LIN {X 0,Y 362.029,Z 234.39,A -85,B 0,C 180,E1 -12949.938,E2 -12949.938} C_VEL
LIN {X 0,Y 362.149,Z 234.377,A -85,B 0,C 180,E1 -12952.192,E2 -12952.192} C_VEL
LIN {X 0,Y 362.116,Z 234.379,A -85,B 0,C 180,E1 -12954.431,E2 -12954.431} C_VEL
LIN {X 0,Y 362.28,Z 234.357,A -85,B 0,C 180,E1 -12957.776,E2 -12957.776} C_VEL
LIN {X 0,Y 362.423,Z 234.341,A -85,B 0,C 180,E1 -12960,E2 -12960} C_VEL
LIN {X 0,Y 362.28,Z 234.36,A -85,B 0,C 180,E1 -12962.223,E2 -12962.223} C_VEL
LIN {X 0,Y 362.17,Z 234.37,A -85,B 0,C 180,E1 -12966.686,E2 -12966.686} C_VEL
LIN {X 0,Y 362.071,Z 234.381,A -85,B 0,C 180,E1 -12968.933,E2 -12968.933} C_VEL
LIN {X 0,Y 361.958,Z 234.4,A -85,B 0,C 180,E1 -12972.332,E2 -12972.332} C_VEL
LIN {X 0,Y 361.959,Z 234.397,A -85,B 0,C 180,E1 -12974.62,E2 -12974.62} C_VEL
LIN {X 0,Y 361.957,Z 234.4,A -85,B 0,C 180,E1 -12978.099,E2 -12978.099} C_VEL
LIN {X 0,Y 361.89,Z 234.404,A -85,B 0,C 180,E1 -12981.653,E2 -12981.653} C_VEL
LIN {X 0,Y 361.926,Z 234.399,A -85,B 0,C 180,E1 -12985.29,E2 -12985.29} C_VEL
LIN {X 0,Y 361.916,Z 234.401,A -85,B 0,C 180,E1 -12987.778,E2 -12987.778} C_VEL
LIN {X 0,Y 361.844,Z 234.409,A -85,B 0,C 180,E1 -12991.285,E2 -12991.285} C_VEL
LIN {X 0,Y 361.852,Z 234.413,A -85,B 0,C 180,E1 -12994.281,E2 -12994.281} C_VEL
LIN {X 0,Y 361.862,Z 234.407,A -85,B 0,C 180,E1 -12997.223,E2 -12997.223} C_VEL
LIN {X 0,Y 361.834,Z 234.413,A -85,B 0,C 180,E1 -13000.756,E2 -13000.756} C_VEL
LIN {X 0,Y 361.816,Z 234.418,A -85,B 0,C 180,E1 -13004.369,E2 -13004.369} C_VEL
LIN {X 0,Y 361.835,Z 234.41,A -85,B 0,C 180,E1 -13007.568,E2 -13007.568} C_VEL
LIN {X 0,Y 361.869,Z 234.407,A -85,B 0,C 180,E1 -13010.974,E2 -13010.974} C_VEL
LIN {X 0,Y 361.874,Z 234.409,A -85,B 0,C 180,E1 -13014.656,E2 -13014.656} C_VEL
LIN {X 0,Y 361.838,Z 234.415,A -85,B 0,C 180,E1 -13018.371,E2 -13018.371} C_VEL
LIN {X 0,Y 361.919,Z 234.533,A -85,B 0,C 180,E1 -13020.495,E2 -13020.495} C_VEL
LIN {X 0,Y 364.089,Z 244.857,A -85,B 0,C 180,E1 -13023.197,E2 -13023.197} C_VEL
LIN {X 0,Y 365.508,Z 253.131,A -85,B 0,C 180,E1 -13025.279,E2 -13025.279} C_VEL
LIN {X 0,Y 364.772,Z 261.991,A -85,B 0,C 180,E1 -13027.336,E2 -13027.336} C_VEL
LIN {X 0,Y 364.414,Z 265.703,A -85,B 0,C 180,E1 -13028.19,E2 -13028.19} C_VEL
LIN {X 0,Y 369.621,Z 298.526,A -85,B 0,C 180,E1 -13029.181,E2 -13029.181} C_VEL
LIN {X 0,Y 368.296,Z 374.24,A -85,B 0,C 180,E1 -13030.709,E2 -13030.709} C_VEL
LIN {X 0,Y 367.689,Z 387.314,A -85,B 0,C 180,E1 -13031.183,E2 -13031.183} C_VEL
LIN {X 0,Y 366.8,Z 399.96,A -85,B 0,C 180,E1 -13031.859,E2 -13031.859} C_VEL
LIN {X 0,Y 365.939,Z 411.236,A -85,B 0,C 180,E1 -13032.682,E2 -13032.682} C_VEL
LIN {X 0,Y 364.86,Z 422.904,A -85,B 0,C 180,E1 -13033.782,E2 -13033.782} C_VEL
LIN {X 0,Y 363.982,Z 432.341,A -85,B 0,C 180,E1 -13034.892,E2 -13034.892} C_VEL
LIN {X 0,Y 363.055,Z 441.998,A -85,B 0,C 180,E1 -13036.283,E2 -13036.283} C_VEL
LIN {X 0,Y 362.203,Z 449.91,A -85,B 0,C 180,E1 -13037.676,E2 -13037.676} C_VEL
LIN {X 0,Y 361.425,Z 457.628,A -85,B 0,C 180,E1 -13039.355,E2 -13039.355} C_VEL
LIN {X 0,Y 360.913,Z 463.827,A -85,B 0,C 180,E1 -13041.038,E2 -13041.038} C_VEL
LIN {X 0,Y 360.588,Z 468.742,A -85,B 0,C 180,E1 -13042.722,E2 -13042.722} C_VEL
LIN {X 0,Y 360.383,Z 472.518,A -85,B 0,C 180,E1 -13044.405,E2 -13044.405} C_VEL
LIN {X 0,Y 360.364,Z 474.464,A -85,B 0,C 180,E1 -13045.526,E2 -13045.526} C_VEL
LIN {X 0,Y 360.3,Z 475.982,A -85,B 0,C 180,E1 -13046.645,E2 -13046.645} C_VEL
LIN {X 0,Y 360.317,Z 477.708,A -85,B 0,C 180,E1 -13048.883,E2 -13048.883} C_VEL
LIN {X 0,Y 360.359,Z 477.984,A -85,B 0,C 180,E1 -13050,E2 -13050} C_VEL
LIN {X 0,Y 360.302,Z 477.86,A -85,B 0,C 180,E1 -13051.118,E2 -13051.118} C_VEL
LIN {X 0,Y 360.297,Z 476.346,A -85,B 0,C 180,E1 -13053.355,E2 -13053.355} C_VEL
LIN {X 0,Y 360.347,Z 474.995,A -85,B 0,C 180,E1 -13054.475,E2 -13054.475} C_VEL
LIN {X 0,Y 360.378,Z 472.521,A -85,B 0,C 180,E1 -13055.961,E2 -13055.961} C_VEL
LIN {X 0,Y 360.672,Z 468.262,A -85,B 0,C 180,E1 -13057.84,E2 -13057.84} C_VEL
LIN {X 0,Y 361.092,Z 463.255,A -85,B 0,C 180,E1 -13059.523,E2 -13059.523} C_VEL
LIN {X 0,Y 361.706,Z 456.971,A -85,B 0,C 180,E1 -13061.204,E2 -13061.204} C_VEL
LIN {X 0,Y 362.689,Z 449.128,A -85,B 0,C 180,E1 -13062.876,E2 -13062.876} C_VEL
LIN {X 0,Y 363.572,Z 441.13,A -85,B 0,C 180,E1 -13064.268,E2 -13064.268} C_VEL
LIN {X 0,Y 364.586,Z 431.385,A -85,B 0,C 180,E1 -13065.657,E2 -13065.657} C_VEL
LIN {X 0,Y 365.793,Z 420.582,A -85,B 0,C 180,E1 -13066.894,E2 -13066.894} C_VEL
LIN {X 0,Y 366.82,Z 410.08,A -85,B 0,C 180,E1 -13067.851,E2 -13067.851} C_VEL
LIN {X 0,Y 367.955,Z 397.467,A -85,B 0,C 180,E1 -13068.731,E2 -13068.731} C_VEL
LIN {X 0,Y 368.842,Z 384.167,A -85,B 0,C 180,E1 -13069.406,E2 -13069.406} C_VEL
LIN {X 0,Y 369.489,Z 370.423,A -85,B 0,C 180,E1 -13069.841,E2 -13069.841} C_VEL
LIN {X 0,Y 370.705,Z 298.181,A -85,B 0,C 180,E1 -13071.303,E2 -13071.303} C_VEL
LIN {X 0,Y 366.607,Z 273.496,A -85,B 0,C 180,E1 -13072.105,E2 -13072.105} C_VEL
LIN {X 0,Y 364.918,Z 264.825,A -85,B 0,C 180,E1 -13072.438,E2 -13072.438} C_VEL
LIN {X 0,Y 365.842,Z 254.94,A -85,B 0,C 180,E1 -13074.698,E2 -13074.698} C_VEL
LIN {X 0,Y 365.142,Z 249.633,A -85,B 0,C 180,E1 -13076.012,E2 -13076.012} C_VEL
LIN {X 0,Y 363.099,Z 239.586,A -85,B 0,C 180,E1 -13078.623,E2 -13078.623} C_VEL
LIN {X 0,Y 361.883,Z 234.409,A -85,B 0,C 180,E1 -13080.023,E2 -13080.023} C_VEL
LIN {X 0,Y 361.86,Z 234.415,A -85,B 0,C 180,E1 -13083.369,E2 -13083.369} C_VEL
LIN {X 0,Y 361.867,Z 234.412,A -85,B 0,C 180,E1 -13087.018,E2 -13087.018} C_VEL
LIN {X 0,Y 361.855,Z 234.408,A -85,B 0,C 180,E1 -13089.861,E2 -13089.861} C_VEL
LIN {X 0,Y 361.837,Z 234.411,A -85,B 0,C 180,E1 -13092.829,E2 -13092.829} C_VEL
LIN {X 0,Y 361.819,Z 234.416,A -85,B 0,C 180,E1 -13095.946,E2 -13095.946} C_VEL
LIN {X 0,Y 361.836,Z 234.415,A -85,B 0,C 180,E1 -13099.244,E2 -13099.244} C_VEL
LIN {X 0,Y 361.863,Z 234.409,A -85,B 0,C 180,E1 -13102.777,E2 -13102.777} C_VEL
LIN {X 0,Y 361.854,Z 234.409,A -85,B 0,C 180,E1 -13105.72,E2 -13105.72} C_VEL
LIN {X 0,Y 361.872,Z 234.407,A -85,B 0,C 180,E1 -13109.672,E2 -13109.672} C_VEL
LIN {X 0,Y 361.954,Z 234.396,A -85,B 0,C 180,E1 -13113.475,E2 -13113.475} C_VEL
LIN {X 0,Y 361.89,Z 234.401,A -85,B 0,C 180,E1 -13117.145,E2 -13117.145} C_VEL
LIN {X 0,Y 361.92,Z 234.399,A -85,B 0,C 180,E1 -13120.724,E2 -13120.724} C_VEL
LIN {X 0,Y 361.945,Z 234.397,A -85,B 0,C 180,E1 -13124.226,E2 -13124.226} C_VEL
LIN {X 0,Y 361.998,Z 234.383,A -85,B 0,C 180,E1 -13126.528,E2 -13126.528} C_VEL
LIN {X 0,Y 362.031,Z 234.381,A -85,B 0,C 180,E1 -13129.938,E2 -13129.938} C_VEL
LIN {X 0,Y 362.16,Z 234.371,A -85,B 0,C 180,E1 -13133.314,E2 -13133.314} C_VEL
LIN {X 0,Y 362.282,Z 234.355,A -85,B 0,C 180,E1 -13137.777,E2 -13137.777} C_VEL
LIN {X 0,Y 362.426,Z 234.33,A -85,B 0,C 180,E1 -13140,E2 -13140} C_VEL
LIN {X 0,Y 362.281,Z 234.357,A -85,B 0,C 180,E1 -13142.224,E2 -13142.224} C_VEL
LIN {X 0,Y 362.17,Z 234.372,A -85,B 0,C 180,E1 -13146.686,E2 -13146.686} C_VEL
LIN {X 0,Y 362.074,Z 234.382,A -85,B 0,C 180,E1 -13148.933,E2 -13148.933} C_VEL
LIN {X 0,Y 361.959,Z 234.392,A -85,B 0,C 180,E1 -13152.332,E2 -13152.332} C_VEL
LIN {X 0,Y 361.962,Z 234.396,A -85,B 0,C 180,E1 -13154.621,E2 -13154.621} C_VEL
LIN {X 0,Y 361.96,Z 234.396,A -85,B 0,C 180,E1 -13158.099,E2 -13158.099} C_VEL
LIN {X 0,Y 361.861,Z 234.408,A -85,B 0,C 180,E1 -13161.655,E2 -13161.655} C_VEL
LIN {X 0,Y 361.901,Z 234.405,A -85,B 0,C 180,E1 -13165.292,E2 -13165.292} C_VEL
LIN {X 0,Y 361.874,Z 234.4,A -85,B 0,C 180,E1 -13169.079,E2 -13169.079} C_VEL
LIN {X 0,Y 361.848,Z 234.411,A -85,B 0,C 180,E1 -13172.945,E2 -13172.945} C_VEL
LIN {X 0,Y 361.867,Z 234.412,A -85,B 0,C 180,E1 -13175.637,E2 -13175.637} C_VEL
LIN {X 0,Y 361.876,Z 234.589,A -85,B 0,C 180,E1 -13179.214,E2 -13179.214} C_VEL
LIN {X 0,Y 364.197,Z 245.232,A -85,B 0,C 180,E1 -13182.112,E2 -13182.112} C_VEL
LIN {X 0,Y 364.641,Z 247.353,A -85,B 0,C 180,E1 -13182.626,E2 -13182.626} C_VEL
LIN {X 0,Y 367.364,Z 255.054,A -85,B 0,C 180,E1 -13182.986,E2 -13182.986} C_VEL
LIN {X 0,Y 371.258,Z 274.03,A -85,B 0,C 180,E1 -13183.657,E2 -13183.657} C_VEL
LIN {X 0,Y 369.515,Z 355.097,A -85,B 0,C 180,E1 -13185.298,E2 -13185.298} C_VEL
LIN {X 0,Y 368.933,Z 368.742,A -85,B 0,C 180,E1 -13185.807,E2 -13185.807} C_VEL
LIN {X 0,Y 368.181,Z 381.251,A -85,B 0,C 180,E1 -13186.499,E2 -13186.499} C_VEL
LIN {X 0,Y 367.234,Z 393.083,A -85,B 0,C 180,E1 -13187.391,E2 -13187.391} C_VEL
LIN {X 0,Y 366.107,Z 405.138,A -85,B 0,C 180,E1 -13188.568,E2 -13188.568} C_VEL
LIN {X 0,Y 364.993,Z 415.361,A -85,B 0,C 180,E1 -13189.832,E2 -13189.832} C_VEL
LIN {X 0,Y 363.968,Z 423.909,A -85,B 0,C 180,E1 -13191.13,E2 -13191.13} C_VEL
LIN {X 0,Y 362.95,Z 432.857,A -85,B 0,C 180,E1 -13192.811,E2 -13192.811} C_VEL
LIN {X 0,Y 362.12,Z 439.647,A -85,B 0,C 180,E1 -13194.392,E2 -13194.392} C_VEL
LIN {X 0,Y 361.357,Z 446.052,A -85,B 0,C 180,E1 -13196.277,E2 -13196.277} C_VEL
LIN {X 0,Y 360.866,Z 451.154,A -85,B 0,C 180,E1 -13198.276,E2 -13198.276} C_VEL
LIN {X 0,Y 360.624,Z 453.662,A -85,B 0,C 180,E1 -13199.556,E2 -13199.556} C_VEL
LIN {X 0,Y 360.339,Z 456.193,A -85,B 0,C 180,E1 -13201.364,E2 -13201.364} C_VEL
LIN {X 0,Y 360.124,Z 457.717,A -85,B 0,C 180,E1 -13203.33,E2 -13203.33} C_VEL
LIN {X 0,Y 360.085,Z 458.053,A -85,B 0,C 180,E1 -13204.571,E2 -13204.571} C_VEL
LIN {X 0,Y 360.06,Z 457.594,A -85,B 0,C 180,E1 -13206.549,E2 -13206.549} C_VEL
LIN {X 0,Y 360.208,Z 456.184,A -85,B 0,C 180,E1 -13208.241,E2 -13208.241} C_VEL
LIN {X 0,Y 360.519,Z 453.638,A -85,B 0,C 180,E1 -13210.053,E2 -13210.053} C_VEL
LIN {X 0,Y 360.83,Z 449.998,A -85,B 0,C 180,E1 -13211.842,E2 -13211.842} C_VEL
LIN {X 0,Y 361.209,Z 445.164,A -85,B 0,C 180,E1 -13213.613,E2 -13213.613} C_VEL
LIN {X 0,Y 361.808,Z 438.966,A -85,B 0,C 180,E1 -13215.373,E2 -13215.373} C_VEL
LIN {X 0,Y 362.631,Z 431.207,A -85,B 0,C 180,E1 -13217.122,E2 -13217.122} C_VEL
LIN {X 0,Y 363.465,Z 423.268,A -85,B 0,C 180,E1 -13218.568,E2 -13218.568} C_VEL
LIN {X 0,Y 364.469,Z 413.538,A -85,B 0,C 180,E1 -13220.006,E2 -13220.006} C_VEL
LIN {X 0,Y 365.519,Z 402.66,A -85,B 0,C 180,E1 -13221.291,E2 -13221.291} C_VEL
LIN {X 0,Y 366.484,Z 392.105,A -85,B 0,C 180,E1 -13222.285,E2 -13222.285} C_VEL
LIN {X 0,Y 367.251,Z 380.768,A -85,B 0,C 180,E1 -13223.131,E2 -13223.131} C_VEL
LIN {X 0,Y 367.916,Z 368.075,A -85,B 0,C 180,E1 -13223.828,E2 -13223.828} C_VEL
LIN {X 0,Y 368.443,Z 354.712,A -85,B 0,C 180,E1 -13224.321,E2 -13224.321} C_VEL
LIN {X 0,Y 369.856,Z 272.512,A -85,B 0,C 180,E1 -13225.982,E2 -13225.982} C_VEL
LIN {X 0,Y 365.244,Z 249.773,A -85,B 0,C 180,E1 -13226.725,E2 -13226.725} C_VEL
LIN {X 0,Y 364.343,Z 246.957,A -85,B 0,C 180,E1 -13226.855,E2 -13226.855} C_VEL
LIN {X 0,Y 363.165,Z 239.521,A -85,B 0,C 180,E1 -13228.891,E2 -13228.891} C_VEL
LIN {X 0,Y 362.19,Z 234.367,A -85,B 0,C 180,E1 -13230.347,E2 -13230.347} C_VEL
LIN {X 0,Y 362.268,Z 234.36,A -85,B 0,C 180,E1 -13232.223,E2 -13232.223} C_VEL
LIN {X 0,Y 362.125,Z 234.374,A -85,B 0,C 180,E1 -13236.687,E2 -13236.687} C_VEL
LIN {X 0,Y 362.048,Z 234.383,A -85,B 0,C 180,E1 -13238.934,E2 -13238.934} C_VEL
LIN {X 0,Y 361.325,Z 234.479,A -85,B 0,C 180,E1 -13239.862,E2 -13239.862} C_VEL
LIN {X 0,Y 358.466,Z 234.835,A -85,B 0,C 180,E1 -13241.37,E2 -13241.37} C_VEL
LIN {X 0,Y 356.073,Z 235.136,A -85,B 0,C 180,E1 -13242.59,E2 -13242.59} C_VEL
LIN {X 0,Y 355.039,Z 235.263,A -85,B 0,C 180,E1 -13243.534,E2 -13243.534} C_VEL
LIN {X 0,Y 354.95,Z 235.272,A -85,B 0,C 180,E1 -13243.853,E2 -13243.853} C_VEL
LIN {X 0,Y 354.925,Z 235.274,A -85,B 0,C 180,E1 -13248.108,E2 -13248.108} C_VEL
LIN {X 0,Y 354.828,Z 235.286,A -85,B 0,C 180,E1 -13252.106,E2 -13252.106} C_VEL
LIN {X 0,Y 354.852,Z 235.286,A -85,B 0,C 180,E1 -13255.831,E2 -13255.831} C_VEL
LIN {X 0,Y 354.8,Z 235.29,A -85,B 0,C 180,E1 -13259.683,E2 -13259.683} C_VEL
LIN {X 0,Y 354.788,Z 235.29,A -85,B 0,C 180,E1 -13262.333,E2 -13262.333} C_VEL
LIN {X 0,Y 354.822,Z 235.288,A -85,B 0,C 180,E1 -13265.699,E2 -13265.699} C_VEL
LIN {X 0,Y 354.824,Z 235.285,A -85,B 0,C 180,E1 -13269.423,E2 -13269.423} C_VEL
LIN {X 0,Y 354.786,Z 235.288,A -85,B 0,C 180,E1 -13272.866,E2 -13272.866} C_VEL
LIN {X 0,Y 354.766,Z 235.295,A -85,B 0,C 180,E1 -13276.103,E2 -13276.103} C_VEL
LIN {X 0,Y 354.786,Z 235.288,A -85,B 0,C 180,E1 -13279.178,E2 -13279.178} C_VEL
LIN {X 0,Y 354.806,Z 235.288,A -85,B 0,C 180,E1 -13282.402,E2 -13282.402} C_VEL
LIN {X 0,Y 354.81,Z 235.285,A -85,B 0,C 180,E1 -13284.94,E2 -13284.94} C_VEL
LIN {X 0,Y 354.792,Z 235.29,A -85,B 0,C 180,E1 -13288.405,E2 -13288.405} C_VEL
LIN {X 0,Y 354.845,Z 235.283,A -85,B 0,C 180,E1 -13291.618,E2 -13291.618} C_VEL
LIN {X 0,Y 354.897,Z 235.279,A -85,B 0,C 180,E1 -13294.172,E2 -13294.172} C_VEL
LIN {X 0,Y 354.833,Z 235.287,A -85,B 0,C 180,E1 -13297.894,E2 -13297.894} C_VEL
LIN {X 0,Y 354.92,Z 235.276,A -85,B 0,C 180,E1 -13301.891,E2 -13301.891} C_VEL
LIN {X 0,Y 354.94,Z 235.274,A -85,B 0,C 180,E1 -13305.981,E2 -13305.981} C_VEL
LIN {X 0,Y 354.976,Z 235.267,A -85,B 0,C 180,E1 -13309.736,E2 -13309.736} C_VEL
LIN {X 0,Y 355.112,Z 235.253,A -85,B 0,C 180,E1 -13312.037,E2 -13312.037} C_VEL
LIN {X 0,Y 355.09,Z 235.255,A -85,B 0,C 180,E1 -13314.321,E2 -13314.321} C_VEL
LIN {X 0,Y 355.243,Z 235.233,A -85,B 0,C 180,E1 -13317.732,E2 -13317.732} C_VEL
LIN {X 0,Y 355.393,Z 235.217,A -85,B 0,C 180,E1 -13320,E2 -13320} C_VEL
LIN {X 0,Y 355.243,Z 235.237,A -85,B 0,C 180,E1 -13322.268,E2 -13322.268} C_VEL
LIN {X 0,Y 355.136,Z 235.245,A -85,B 0,C 180,E1 -13326.819,E2 -13326.819} C_VEL
LIN {X 0,Y 355.013,Z 235.26,A -85,B 0,C 180,E1 -13329.112,E2 -13329.112} C_VEL
LIN {X 0,Y 354.919,Z 235.274,A -85,B 0,C 180,E1 -13332.581,E2 -13332.581} C_VEL
LIN {X 0,Y 354.887,Z 235.28,A -85,B 0,C 180,E1 -13336.096,E2 -13336.096} C_VEL
LIN {X 0,Y 354.904,Z 235.278,A -85,B 0,C 180,E1 -13338.472,E2 -13338.472} C_VEL
LIN {X 0,Y 354.832,Z 235.287,A -85,B 0,C 180,E1 -13342.106,E2 -13342.106} C_VEL
LIN {X 0,Y 354.897,Z 235.276,A -85,B 0,C 180,E1 -13345.828,E2 -13345.828} C_VEL
LIN {X 0,Y 354.852,Z 235.28,A -85,B 0,C 180,E1 -13349.679,E2 -13349.679} C_VEL
LIN {X 0,Y 354.804,Z 235.286,A -85,B 0,C 180,E1 -13353.702,E2 -13353.702} C_VEL
LIN {X 0,Y 354.797,Z 235.292,A -85,B 0,C 180,E1 -13356.46,E2 -13356.46} C_VEL
LIN {X 0,Y 354.822,Z 235.283,A -85,B 0,C 180,E1 -13359.424,E2 -13359.424} C_VEL
LIN {X 0,Y 354.786,Z 235.29,A -85,B 0,C 180,E1 -13362.868,E2 -13362.868} C_VEL
LIN {X 0,Y 354.766,Z 235.294,A -85,B 0,C 180,E1 -13366.104,E2 -13366.104} C_VEL
LIN {X 0,Y 354.787,Z 235.288,A -85,B 0,C 180,E1 -13369.179,E2 -13369.179} C_VEL
LIN {X 0,Y 354.81,Z 235.291,A -85,B 0,C 180,E1 -13372.402,E2 -13372.402} C_VEL
LIN {X 0,Y 354.811,Z 235.286,A -85,B 0,C 180,E1 -13374.941,E2 -13374.941} C_VEL
LIN {X 0,Y 354.793,Z 235.293,A -85,B 0,C 180,E1 -13378.405,E2 -13378.405} C_VEL
LIN {X 0,Y 354.871,Z 235.377,A -85,B 0,C 180,E1 -13380.16,E2 -13380.16} C_VEL
LIN {X 0,Y 357.175,Z 246.354,A -85,B 0,C 180,E1 -13383.092,E2 -13383.092} C_VEL
LIN {X 0,Y 358.515,Z 254.059,A -85,B 0,C 180,E1 -13385.073,E2 -13385.073} C_VEL
LIN {X 0,Y 357.995,Z 261.662,A -85,B 0,C 180,E1 -13386.882,E2 -13386.882} C_VEL
LIN {X 0,Y 357.535,Z 265.52,A -85,B 0,C 180,E1 -13387.783,E2 -13387.783} C_VEL
LIN {X 0,Y 362.845,Z 298.374,A -85,B 0,C 180,E1 -13388.804,E2 -13388.804} C_VEL
LIN {X 0,Y 361.735,Z 368.666,A -85,B 0,C 180,E1 -13390.234,E2 -13390.234} C_VEL
LIN {X 0,Y 361.18,Z 382.385,A -85,B 0,C 180,E1 -13390.646,E2 -13390.646} C_VEL
LIN {X 0,Y 360.411,Z 394.736,A -85,B 0,C 180,E1 -13391.232,E2 -13391.232} C_VEL
LIN {X 0,Y 359.636,Z 405.389,A -85,B 0,C 180,E1 -13391.927,E2 -13391.927} C_VEL
LIN {X 0,Y 358.569,Z 416.918,A -85,B 0,C 180,E1 -13392.903,E2 -13392.903} C_VEL
LIN {X 0,Y 357.4,Z 428.473,A -85,B 0,C 180,E1 -13394.153,E2 -13394.153} C_VEL
LIN {X 0,Y 356.531,Z 438.002,A -85,B 0,C 180,E1 -13395.444,E2 -13395.444} C_VEL
LIN {X 0,Y 355.606,Z 446.571,A -85,B 0,C 180,E1 -13396.863,E2 -13396.863} C_VEL
LIN {X 0,Y 354.604,Z 454.901,A -85,B 0,C 180,E1 -13398.569,E2 -13398.569} C_VEL
LIN {X 0,Y 354.018,Z 461.619,A -85,B 0,C 180,E1 -13400.286,E2 -13400.286} C_VEL
LIN {X 0,Y 353.609,Z 466.972,A -85,B 0,C 180,E1 -13402.003,E2 -13402.003} C_VEL
LIN {X 0,Y 353.314,Z 471.786,A -85,B 0,C 180,E1 -13404.035,E2 -13404.035} C_VEL
LIN {X 0,Y 353.277,Z 474.224,A -85,B 0,C 180,E1 -13405.436,E2 -13405.436} C_VEL
LIN {X 0,Y 353.222,Z 475.755,A -85,B 0,C 180,E1 -13406.578,E2 -13406.578} C_VEL
LIN {X 0,Y 353.217,Z 477.5,A -85,B 0,C 180,E1 -13408.86,E2 -13408.86} C_VEL
LIN {X 0,Y 353.262,Z 477.783,A -85,B 0,C 180,E1 -13410,E2 -13410} C_VEL
LIN {X 0,Y 353.202,Z 477.67,A -85,B 0,C 180,E1 -13411.14,E2 -13411.14} C_VEL
LIN {X 0,Y 353.171,Z 477.121,A -85,B 0,C 180,E1 -13412.281,E2 -13412.281} C_VEL
LIN {X 0,Y 353.218,Z 476.174,A -85,B 0,C 180,E1 -13413.422,E2 -13413.422} C_VEL
LIN {X 0,Y 353.26,Z 474.829,A -85,B 0,C 180,E1 -13414.564,E2 -13414.564} C_VEL
LIN {X 0,Y 353.275,Z 472.703,A -85,B 0,C 180,E1 -13415.905,E2 -13415.905} C_VEL
LIN {X 0,Y 353.617,Z 468.125,A -85,B 0,C 180,E1 -13417.997,E2 -13417.997} C_VEL
LIN {X 0,Y 354.057,Z 463.133,A -85,B 0,C 180,E1 -13419.714,E2 -13419.714} C_VEL
LIN {X 0,Y 354.704,Z 456.869,A -85,B 0,C 180,E1 -13421.428,E2 -13421.428} C_VEL
LIN {X 0,Y 355.743,Z 449.067,A -85,B 0,C 180,E1 -13423.132,E2 -13423.132} C_VEL
LIN {X 0,Y 356.653,Z 441.105,A -85,B 0,C 180,E1 -13424.551,E2 -13424.551} C_VEL
LIN {X 0,Y 357.881,Z 430.336,A -85,B 0,C 180,E1 -13426.104,E2 -13426.104} C_VEL
LIN {X 0,Y 359.116,Z 419.292,A -85,B 0,C 180,E1 -13427.364,E2 -13427.364} C_VEL
LIN {X 0,Y 360.277,Z 408.49,A -85,B 0,C 180,E1 -13428.334,E2 -13428.334} C_VEL
LIN {X 0,Y 361.361,Z 396.619,A -85,B 0,C 180,E1 -13429.159,E2 -13429.159} C_VEL
LIN {X 0,Y 362.214,Z 383.848,A -85,B 0,C 180,E1 -13429.813,E2 -13429.813} C_VEL
LIN {X 0,Y 362.886,Z 370.019,A -85,B 0,C 180,E1 -13430.254,E2 -13430.254} C_VEL
LIN {X 0,Y 364.227,Z 299.716,A -85,B 0,C 180,E1 -13431.697,E2 -13431.697} C_VEL
LIN {X 0,Y 360.413,Z 276.099,A -85,B 0,C 180,E1 -13432.48,E2 -13432.48} C_VEL
LIN {X 0,Y 358.119,Z 264.715,A -85,B 0,C 180,E1 -13432.905,E2 -13432.905} C_VEL
LIN {X 0,Y 358.954,Z 256.182,A -85,B 0,C 180,E1 -13434.895,E2 -13434.895} C_VEL
LIN {X 0,Y 357.778,Z 248.514,A -85,B 0,C 180,E1 -13436.859,E2 -13436.859} C_VEL
LIN {X 0,Y 355.535,Z 238.291,A -85,B 0,C 180,E1 -13439.616,E2 -13439.616} C_VEL
LIN {X 0,Y 354.84,Z 235.286,A -85,B 0,C 180,E1 -13440.499,E2 -13440.499} C_VEL
LIN {X 0,Y 354.807,Z 235.293,A -85,B 0,C 180,E1 -13443.702,E2 -13443.702} C_VEL
LIN {X 0,Y 354.798,Z 235.289,A -85,B 0,C 180,E1 -13446.459,E2 -13446.459} C_VEL
LIN {X 0,Y 354.825,Z 235.286,A -85,B 0,C 180,E1 -13449.423,E2 -13449.423} C_VEL
LIN {X 0,Y 354.789,Z 235.289,A -85,B 0,C 180,E1 -13452.867,E2 -13452.867} C_VEL
LIN {X 0,Y 354.768,Z 235.294,A -85,B 0,C 180,E1 -13456.104,E2 -13456.104} C_VEL
LIN {X 0,Y 354.788,Z 235.292,A -85,B 0,C 180,E1 -13459.179,E2 -13459.179} C_VEL
LIN {X 0,Y 354.807,Z 235.286,A -85,B 0,C 180,E1 -13462.402,E2 -13462.402} C_VEL
LIN {X 0,Y 354.812,Z 235.283,A -85,B 0,C 180,E1 -13464.941,E2 -13464.941} C_VEL
LIN {X 0,Y 354.793,Z 235.284,A -85,B 0,C 180,E1 -13468.405,E2 -13468.405} C_VEL
LIN {X 0,Y 354.846,Z 235.279,A -85,B 0,C 180,E1 -13471.619,E2 -13471.619} C_VEL
LIN {X 0,Y 354.899,Z 235.274,A -85,B 0,C 180,E1 -13474.173,E2 -13474.173} C_VEL
LIN {X 0,Y 354.834,Z 235.281,A -85,B 0,C 180,E1 -13477.894,E2 -13477.894} C_VEL
LIN {X 0,Y 354.923,Z 235.267,A -85,B 0,C 180,E1 -13481.891,E2 -13481.891} C_VEL
LIN {X 0,Y 354.942,Z 235.26,A -85,B 0,C 180,E1 -13485.981,E2 -13485.981} C_VEL
LIN {X 0,Y 354.978,Z 235.26,A -85,B 0,C 180,E1 -13489.736,E2 -13489.736} C_VEL
LIN {X 0,Y 355.124,Z 235.248,A -85,B 0,C 180,E1 -13493.181,E2 -13493.181} C_VEL
LIN {X 0,Y 355.245,Z 235.232,A -85,B 0,C 180,E1 -13497.732,E2 -13497.732} C_VEL
LIN {X 0,Y 355.374,Z 235.208,A -85,B 0,C 180,E1 -13500,E2 -13500} C_VEL
LIN {X 0,Y 355.244,Z 235.234,A -85,B 0,C 180,E1 -13502.268,E2 -13502.268} C_VEL
LIN {X 0,Y 355.136,Z 235.246,A -85,B 0,C 180,E1 -13506.819,E2 -13506.819} C_VEL
LIN {X 0,Y 355.015,Z 235.263,A -85,B 0,C 180,E1 -13509.112,E2 -13509.112} C_VEL
LIN {X 0,Y 354.92,Z 235.271,A -85,B 0,C 180,E1 -13512.581,E2 -13512.581} C_VEL
LIN {X 0,Y 354.89,Z 235.275,A -85,B 0,C 180,E1 -13516.096,E2 -13516.096} C_VEL
LIN {X 0,Y 354.906,Z 235.274,A -85,B 0,C 180,E1 -13518.472,E2 -13518.472} C_VEL
LIN {X 0,Y 354.815,Z 235.287,A -85,B 0,C 180,E1 -13522.108,E2 -13522.108} C_VEL
LIN {X 0,Y 354.863,Z 235.281,A -85,B 0,C 180,E1 -13525.83,E2 -13525.83} C_VEL
LIN {X 0,Y 354.807,Z 235.283,A -85,B 0,C 180,E1 -13529.683,E2 -13529.683} C_VEL
LIN {X 0,Y 354.814,Z 235.291,A -85,B 0,C 180,E1 -13533.684,E2 -13533.684} C_VEL
LIN {X 0,Y 354.796,Z 235.296,A -85,B 0,C 180,E1 -13536.46,E2 -13536.46} C_VEL
LIN {X 0,Y 354.835,Z 235.444,A -85,B 0,C 180,E1 -13538.784,E2 -13538.784} C_VEL
LIN {X 0,Y 357.046,Z 245.454,A -85,B 0,C 180,E1 -13541.584,E2 -13541.584} C_VEL
LIN {X 0,Y 357.421,Z 247.366,A -85,B 0,C 180,E1 -13542.097,E2 -13542.097} C_VEL
LIN {X 0,Y 361.007,Z 256.704,A -85,B 0,C 180,E1 -13542.571,E2 -13542.571} C_VEL
LIN {X 0,Y 364.664,Z 274.592,A -85,B 0,C 180,E1 -13543.225,E2 -13543.225} C_VEL
LIN {X 0,Y 362.909,Z 355.501,A -85,B 0,C 180,E1 -13544.898,E2 -13544.898} C_VEL
LIN {X 0,Y 362.308,Z 369.069,A -85,B 0,C 180,E1 -13545.416,E2 -13545.416} C_VEL
LIN {X 0,Y 361.56,Z 381.138,A -85,B 0,C 180,E1 -13546.094,E2 -13546.094} C_VEL
LIN {X 0,Y 360.586,Z 392.893,A -85,B 0,C 180,E1 -13546.987,E2 -13546.987} C_VEL
LIN {X 0,Y 359.475,Z 404.017,A -85,B 0,C 180,E1 -13548.073,E2 -13548.073} C_VEL
LIN {X 0,Y 358.374,Z 414.089,A -85,B 0,C 180,E1 -13549.303,E2 -13549.303} C_VEL
LIN {X 0,Y 357.247,Z 423.071,A -85,B 0,C 180,E1 -13550.648,E2 -13550.648} C_VEL
LIN {X 0,Y 356.158,Z 431.861,A -85,B 0,C 180,E1 -13552.286,E2 -13552.286} C_VEL
LIN {X 0,Y 355.228,Z 439.149,A -85,B 0,C 180,E1 -13553.973,E2 -13553.973} C_VEL
LIN {X 0,Y 354.559,Z 444.812,A -85,B 0,C 180,E1 -13555.603,E2 -13555.603} C_VEL
LIN {X 0,Y 353.97,Z 450.193,A -85,B 0,C 180,E1 -13557.583,E2 -13557.583} C_VEL
LIN {X 0,Y 353.557,Z 454.052,A -85,B 0,C 180,E1 -13559.543,E2 -13559.543} C_VEL
LIN {X 0,Y 353.22,Z 456.598,A -85,B 0,C 180,E1 -13561.476,E2 -13561.476} C_VEL
LIN {X 0,Y 353.037,Z 458.056,A -85,B 0,C 180,E1 -13563.616,E2 -13563.616} C_VEL
LIN {X 0,Y 352.975,Z 458.214,A -85,B 0,C 180,E1 -13565.284,E2 -13565.284} C_VEL
LIN {X 0,Y 352.986,Z 457.797,A -85,B 0,C 180,E1 -13566.534,E2 -13566.534} C_VEL
LIN {X 0,Y 353.049,Z 456.88,A -85,B 0,C 180,E1 -13567.776,E2 -13567.776} C_VEL
LIN {X 0,Y 353.256,Z 455.198,A -85,B 0,C 180,E1 -13569.239,E2 -13569.239} C_VEL
LIN {X 0,Y 353.556,Z 452.507,A -85,B 0,C 180,E1 -13570.853,E2 -13570.853} C_VEL
LIN {X 0,Y 353.899,Z 448.408,A -85,B 0,C 180,E1 -13572.67,E2 -13572.67} C_VEL
LIN {X 0,Y 354.391,Z 443.078,A -85,B 0,C 180,E1 -13574.471,E2 -13574.471} C_VEL
LIN {X 0,Y 355.148,Z 436.271,A -85,B 0,C 180,E1 -13576.263,E2 -13576.263} C_VEL
LIN {X 0,Y 356.062,Z 427.788,A -85,B 0,C 180,E1 -13578.039,E2 -13578.039} C_VEL
LIN {X 0,Y 357.047,Z 418.879,A -85,B 0,C 180,E1 -13579.538,E2 -13579.538} C_VEL
LIN {X 0,Y 358.137,Z 408.245,A -85,B 0,C 180,E1 -13580.968,E2 -13580.968} C_VEL
LIN {X 0,Y 359.21,Z 397.431,A -85,B 0,C 180,E1 -13582.128,E2 -13582.128} C_VEL
LIN {X 0,Y 360.112,Z 385.532,A -85,B 0,C 180,E1 -13583.135,E2 -13583.135} C_VEL
LIN {X 0,Y 360.941,Z 372.334,A -85,B 0,C 180,E1 -13583.961,E2 -13583.961} C_VEL
LIN {X 0,Y 361.596,Z 359.31,A -85,B 0,C 180,E1 -13584.526,E2 -13584.526} C_VEL
LIN {X 0,Y 361.952,Z 345.769,A -85,B 0,C 180,E1 -13584.876,E2 -13584.876} C_VEL
LIN {X 0,Y 363.24,Z 273.905,A -85,B 0,C 180,E1 -13586.327,E2 -13586.327} C_VEL
LIN {X 0,Y 358.907,Z 252.288,A -85,B 0,C 180,E1 -13587.046,E2 -13587.046} C_VEL
LIN {X 0,Y 357.253,Z 247.11,A -85,B 0,C 180,E1 -13587.285,E2 -13587.285} C_VEL
LIN {X 0,Y 355.954,Z 239.449,A -85,B 0,C 180,E1 -13589.434,E2 -13589.434} C_VEL
LIN {X 0,Y 355.15,Z 235.247,A -85,B 0,C 180,E1 -13590.708,E2 -13590.708} C_VEL
LIN {X 0,Y 355.23,Z 235.237,A -85,B 0,C 180,E1 -13592.268,E2 -13592.268} C_VEL
LIN {X 0,Y 355.091,Z 235.25,A -85,B 0,C 180,E1 -13596.82,E2 -13596.82} C_VEL
LIN {X 0,Y 354.958,Z 235.268,A -85,B 0,C 180,E1 -13600.264,E2 -13600.264} C_VEL
LIN {X 0,Y 354.95,Z 235.272,A -85,B 0,C 180,E1 -13603.853,E2 -13603.853} C_VEL
LIN {X 0,Y 354.277,Z 235.353,A -85,B 0,C 180,E1 -13604.799,E2 -13604.799} C_VEL
LIN {X 0,Y 351.451,Z 235.706,A -85,B 0,C 180,E1 -13606.338,E2 -13606.338} C_VEL
LIN {X 0,Y 349.037,Z 236.008,A -85,B 0,C 180,E1 -13607.584,E2 -13607.584} C_VEL
LIN {X 0,Y 347.961,Z 236.139,A -85,B 0,C 180,E1 -13608.546,E2 -13608.546} C_VEL
LIN {X 0,Y 347.851,Z 236.151,A -85,B 0,C 180,E1 -13608.873,E2 -13608.873} C_VEL
LIN {X 0,Y 347.77,Z 236.162,A -85,B 0,C 180,E1 -13612.579,E2 -13612.579} C_VEL
LIN {X 0,Y 347.787,Z 236.16,A -85,B 0,C 180,E1 -13615.11,E2 -13615.11} C_VEL
LIN {X 0,Y 347.747,Z 236.165,A -85,B 0,C 180,E1 -13619.015,E2 -13619.015} C_VEL
LIN {X 0,Y 347.74,Z 236.172,A -85,B 0,C 180,E1 -13621.914,E2 -13621.914} C_VEL
LIN {X 0,Y 347.788,Z 236.165,A -85,B 0,C 180,E1 -13625.875,E2 -13625.875} C_VEL
LIN {X 0,Y 347.751,Z 236.164,A -85,B 0,C 180,E1 -13628.792,E2 -13628.792} C_VEL
LIN {X 0,Y 347.748,Z 236.17,A -85,B 0,C 180,E1 -13631.83,E2 -13631.83} C_VEL
LIN {X 0,Y 347.705,Z 236.17,A -85,B 0,C 180,E1 -13635.026,E2 -13635.026} C_VEL
LIN {X 0,Y 347.749,Z 236.166,A -85,B 0,C 180,E1 -13638.397,E2 -13638.397} C_VEL
LIN {X 0,Y 347.772,Z 236.168,A -85,B 0,C 180,E1 -13642.011,E2 -13642.011} C_VEL
LIN {X 0,Y 347.743,Z 236.167,A -85,B 0,C 180,E1 -13645.536,E2 -13645.536} C_VEL
LIN {X 0,Y 347.743,Z 236.168,A -85,B 0,C 180,E1 -13648.3,E2 -13648.3} C_VEL
LIN {X 0,Y 347.777,Z 236.161,A -85,B 0,C 180,E1 -13650.987,E2 -13650.987} C_VEL
LIN {X 0,Y 347.829,Z 236.156,A -85,B 0,C 180,E1 -13653.607,E2 -13653.607} C_VEL
LIN {X 0,Y 347.787,Z 236.165,A -85,B 0,C 180,E1 -13656.162,E2 -13656.162} C_VEL
LIN {X 0,Y 347.812,Z 236.161,A -85,B 0,C 180,E1 -13659.909,E2 -13659.909} C_VEL
LIN {X 0,Y 347.864,Z 236.154,A -85,B 0,C 180,E1 -13662.359,E2 -13662.359} C_VEL
LIN {X 0,Y 347.895,Z 236.151,A -85,B 0,C 180,E1 -13665.971,E2 -13665.971} C_VEL
LIN {X 0,Y 347.926,Z 236.143,A -85,B 0,C 180,E1 -13669.525,E2 -13669.525} C_VEL
LIN {X 0,Y 348.072,Z 236.128,A -85,B 0,C 180,E1 -13671.875,E2 -13671.875} C_VEL
LIN {X 0,Y 348.065,Z 236.131,A -85,B 0,C 180,E1 -13674.206,E2 -13674.206} C_VEL
LIN {X 0,Y 348.206,Z 236.109,A -85,B 0,C 180,E1 -13677.686,E2 -13677.686} C_VEL
LIN {X 0,Y 348.342,Z 236.095,A -85,B 0,C 180,E1 -13680,E2 -13680} C_VEL
LIN {X 0,Y 348.206,Z 236.113,A -85,B 0,C 180,E1 -13682.313,E2 -13682.313} C_VEL
LIN {X 0,Y 348.104,Z 236.12,A -85,B 0,C 180,E1 -13686.958,E2 -13686.958} C_VEL
LIN {X 0,Y 347.965,Z 236.137,A -85,B 0,C 180,E1 -13689.299,E2 -13689.299} C_VEL
LIN {X 0,Y 347.887,Z 236.148,A -85,B 0,C 180,E1 -13692.839,E2 -13692.839} C_VEL
LIN {X 0,Y 347.837,Z 236.158,A -85,B 0,C 180,E1 -13696.431,E2 -13696.431} C_VEL
LIN {X 0,Y 347.853,Z 236.152,A -85,B 0,C 180,E1 -13698.86,E2 -13698.86} C_VEL
LIN {X 0,Y 347.772,Z 236.165,A -85,B 0,C 180,E1 -13702.579,E2 -13702.579} C_VEL
LIN {X 0,Y 347.81,Z 236.157,A -85,B 0,C 180,E1 -13705.109,E2 -13705.109} C_VEL
LIN {X 0,Y 347.809,Z 236.158,A -85,B 0,C 180,E1 -13707.694,E2 -13707.694} C_VEL
LIN {X 0,Y 347.761,Z 236.169,A -85,B 0,C 180,E1 -13710.347,E2 -13710.347} C_VEL
LIN {X 0,Y 347.742,Z 236.17,A -85,B 0,C 180,E1 -13714.464,E2 -13714.464} C_VEL
LIN {X 0,Y 347.772,Z 236.164,A -85,B 0,C 180,E1 -13717.989,E2 -13717.989} C_VEL
LIN {X 0,Y 347.749,Z 236.166,A -85,B 0,C 180,E1 -13721.831,E2 -13721.831} C_VEL
LIN {X 0,Y 347.704,Z 236.171,A -85,B 0,C 180,E1 -13725.027,E2 -13725.027} C_VEL
LIN {X 0,Y 347.749,Z 236.171,A -85,B 0,C 180,E1 -13728.398,E2 -13728.398} C_VEL
LIN {X 0,Y 347.775,Z 236.163,A -85,B 0,C 180,E1 -13732.011,E2 -13732.011} C_VEL
LIN {X 0,Y 347.744,Z 236.165,A -85,B 0,C 180,E1 -13735.537,E2 -13735.537} C_VEL
LIN {X 0,Y 347.86,Z 236.345,A -85,B 0,C 180,E1 -13739.847,E2 -13739.847} C_VEL
LIN {X 0,Y 350.138,Z 247.263,A -85,B 0,C 180,E1 -13742.83,E2 -13742.83} C_VEL
LIN {X 0,Y 351.63,Z 256.261,A -85,B 0,C 180,E1 -13745.183,E2 -13745.183} C_VEL
LIN {X 0,Y 350.679,Z 265.344,A -85,B 0,C 180,E1 -13747.365,E2 -13747.365} C_VEL
LIN {X 0,Y 356.201,Z 299.78,A -85,B 0,C 180,E1 -13748.458,E2 -13748.458} C_VEL
LIN {X 0,Y 354.805,Z 374.115,A -85,B 0,C 180,E1 -13750.021,E2 -13750.021} C_VEL
LIN {X 0,Y 354.171,Z 387.102,A -85,B 0,C 180,E1 -13750.512,E2 -13750.512} C_VEL
LIN {X 0,Y 353.207,Z 399.702,A -85,B 0,C 180,E1 -13751.211,E2 -13751.211} C_VEL
LIN {X 0,Y 352.208,Z 411.739,A -85,B 0,C 180,E1 -13752.134,E2 -13752.134} C_VEL
LIN {X 0,Y 351.061,Z 423.25,A -85,B 0,C 180,E1 -13753.275,E2 -13753.275} C_VEL
LIN {X 0,Y 350.005,Z 433.435,A -85,B 0,C 180,E1 -13754.543,E2 -13754.543} C_VEL
LIN {X 0,Y 348.974,Z 442.95,A -85,B 0,C 180,E1 -13756.015,E2 -13756.015} C_VEL
LIN {X 0,Y 348.122,Z 450.623,A -85,B 0,C 180,E1 -13757.466,E2 -13757.466} C_VEL
LIN {X 0,Y 347.285,Z 458.135,A -85,B 0,C 180,E1 -13759.211,E2 -13759.211} C_VEL
LIN {X 0,Y 346.678,Z 465.064,A -85,B 0,C 180,E1 -13761.255,E2 -13761.255} C_VEL
LIN {X 0,Y 346.341,Z 469.622,A -85,B 0,C 180,E1 -13763.007,E2 -13763.007} C_VEL
LIN {X 0,Y 346.201,Z 472.02,A -85,B 0,C 180,E1 -13764.175,E2 -13764.175} C_VEL
LIN {X 0,Y 346.173,Z 473.984,A -85,B 0,C 180,E1 -13765.342,E2 -13765.342} C_VEL
LIN {X 0,Y 346.145,Z 475.527,A -85,B 0,C 180,E1 -13766.508,E2 -13766.508} C_VEL
LIN {X 0,Y 346.084,Z 476.611,A -85,B 0,C 180,E1 -13767.673,E2 -13767.673} C_VEL
LIN {X 0,Y 346.117,Z 477.292,A -85,B 0,C 180,E1 -13768.837,E2 -13768.837} C_VEL
LIN {X 0,Y 346.164,Z 477.582,A -85,B 0,C 180,E1 -13770,E2 -13770} C_VEL
LIN {X 0,Y 346.103,Z 477.478,A -85,B 0,C 180,E1 -13771.164,E2 -13771.164} C_VEL
LIN {X 0,Y 346.083,Z 476.942,A -85,B 0,C 180,E1 -13772.328,E2 -13772.328} C_VEL
LIN {X 0,Y 346.141,Z 476.002,A -85,B 0,C 180,E1 -13773.492,E2 -13773.492} C_VEL
LIN {X 0,Y 346.158,Z 474.664,A -85,B 0,C 180,E1 -13774.658,E2 -13774.658} C_VEL
LIN {X 0,Y 346.241,Z 471.844,A -85,B 0,C 180,E1 -13776.409,E2 -13776.409} C_VEL
LIN {X 0,Y 346.557,Z 467.998,A -85,B 0,C 180,E1 -13778.161,E2 -13778.161} C_VEL
LIN {X 0,Y 347.039,Z 463.03,A -85,B 0,C 180,E1 -13779.912,E2 -13779.912} C_VEL
LIN {X 0,Y 347.716,Z 456.79,A -85,B 0,C 180,E1 -13781.661,E2 -13781.661} C_VEL
LIN {X 0,Y 348.804,Z 449.027,A -85,B 0,C 180,E1 -13783.398,E2 -13783.398} C_VEL
LIN {X 0,Y 349.756,Z 441.096,A -85,B 0,C 180,E1 -13784.845,E2 -13784.845} C_VEL
LIN {X 0,Y 351.055,Z 430.362,A -85,B 0,C 180,E1 -13786.426,E2 -13786.426} C_VEL
LIN {X 0,Y 352.366,Z 419.393,A -85,B 0,C 180,E1 -13787.708,E2 -13787.708} C_VEL
LIN {X 0,Y 353.735,Z 406.898,A -85,B 0,C 180,E1 -13788.836,E2 -13788.836} C_VEL
LIN {X 0,Y 354.879,Z 394.64,A -85,B 0,C 180,E1 -13789.674,E2 -13789.674} C_VEL
LIN {X 0,Y 355.772,Z 381.735,A -85,B 0,C 180,E1 -13790.3,E2 -13790.3} C_VEL
LIN {X 0,Y 356.373,Z 368.15,A -85,B 0,C 180,E1 -13790.717,E2 -13790.717} C_VEL
LIN {X 0,Y 357.597,Z 299.819,A -85,B 0,C 180,E1 -13792.151,E2 -13792.151} C_VEL
LIN {X 0,Y 354.011,Z 277.565,A -85,B 0,C 180,E1 -13792.913,E2 -13792.913} C_VEL
LIN {X 0,Y 351.356,Z 264.399,A -85,B 0,C 180,E1 -13793.441,E2 -13793.441} C_VEL
LIN {X 0,Y 352.086,Z 257.528,A -85,B 0,C 180,E1 -13795.077,E2 -13795.077} C_VEL
LIN {X 0,Y 350.609,Z 248.498,A -85,B 0,C 180,E1 -13797.454,E2 -13797.454} C_VEL
LIN {X 0,Y 347.943,Z 236.996,A -85,B 0,C 180,E1 -13800.665,E2 -13800.665} C_VEL
LIN {X 0,Y 347.78,Z 236.168,A -85,B 0,C 180,E1 -13800.934,E2 -13800.934} C_VEL
LIN {X 0,Y 347.745,Z 236.17,A -85,B 0,C 180,E1 -13804.464,E2 -13804.464} C_VEL
LIN {X 0,Y 347.774,Z 236.163,A -85,B 0,C 180,E1 -13807.988,E2 -13807.988} C_VEL
LIN {X 0,Y 347.751,Z 236.166,A -85,B 0,C 180,E1 -13811.83,E2 -13811.83} C_VEL
LIN {X 0,Y 347.707,Z 236.172,A -85,B 0,C 180,E1 -13815.026,E2 -13815.026} C_VEL
LIN {X 0,Y 347.75,Z 236.162,A -85,B 0,C 180,E1 -13818.397,E2 -13818.397} C_VEL
LIN {X 0,Y 347.773,Z 236.162,A -85,B 0,C 180,E1 -13822.011,E2 -13822.011} C_VEL
LIN {X 0,Y 347.744,Z 236.166,A -85,B 0,C 180,E1 -13825.536,E2 -13825.536} C_VEL
LIN {X 0,Y 347.744,Z 236.162,A -85,B 0,C 180,E1 -13828.3,E2 -13828.3} C_VEL
LIN {X 0,Y 347.779,Z 236.166,A -85,B 0,C 180,E1 -13830.988,E2 -13830.988} C_VEL
LIN {X 0,Y 347.831,Z 236.156,A -85,B 0,C 180,E1 -13833.608,E2 -13833.608} C_VEL
LIN {X 0,Y 347.788,Z 236.158,A -85,B 0,C 180,E1 -13836.162,E2 -13836.162} C_VEL
LIN {X 0,Y 347.817,Z 236.156,A -85,B 0,C 180,E1 -13839.91,E2 -13839.91} C_VEL
LIN {X 0,Y 347.866,Z 236.147,A -85,B 0,C 180,E1 -13842.359,E2 -13842.359} C_VEL
LIN {X 0,Y 347.897,Z 236.137,A -85,B 0,C 180,E1 -13845.971,E2 -13845.971} C_VEL
LIN {X 0,Y 347.928,Z 236.139,A -85,B 0,C 180,E1 -13849.526,E2 -13849.526} C_VEL
LIN {X 0,Y 348.091,Z 236.126,A -85,B 0,C 180,E1 -13853.042,E2 -13853.042} C_VEL
LIN {X 0,Y 348.207,Z 236.109,A -85,B 0,C 180,E1 -13857.687,E2 -13857.687} C_VEL
LIN {X 0,Y 348.325,Z 236.086,A -85,B 0,C 180,E1 -13860,E2 -13860} C_VEL
LIN {X 0,Y 348.207,Z 236.111,A -85,B 0,C 180,E1 -13862.314,E2 -13862.314} C_VEL
LIN {X 0,Y 348.105,Z 236.121,A -85,B 0,C 180,E1 -13866.958,E2 -13866.958} C_VEL
LIN {X 0,Y 347.967,Z 236.14,A -85,B 0,C 180,E1 -13869.299,E2 -13869.299} C_VEL
LIN {X 0,Y 347.889,Z 236.15,A -85,B 0,C 180,E1 -13872.84,E2 -13872.84} C_VEL
LIN {X 0,Y 347.839,Z 236.156,A -85,B 0,C 180,E1 -13876.432,E2 -13876.432} C_VEL
LIN {X 0,Y 347.855,Z 236.154,A -85,B 0,C 180,E1 -13878.86,E2 -13878.86} C_VEL
LIN {X 0,Y 347.761,Z 236.17,A -85,B 0,C 180,E1 -13882.58,E2 -13882.58} C_VEL
LIN {X 0,Y 347.792,Z 236.163,A -85,B 0,C 180,E1 -13885.11,E2 -13885.11} C_VEL
LIN {X 0,Y 347.757,Z 236.158,A -85,B 0,C 180,E1 -13889.015,E2 -13889.015} C_VEL
LIN {X 0,Y 347.733,Z 236.17,A -85,B 0,C 180,E1 -13893.072,E2 -13893.072} C_VEL
LIN {X 0,Y 347.769,Z 236.171,A -85,B 0,C 180,E1 -13896.065,E2 -13896.065} C_VEL
LIN {X 0,Y 347.787,Z 236.324,A -85,B 0,C 180,E1 -13898.334,E2 -13898.334} C_VEL
LIN {X 0,Y 349.971,Z 246.018,A -85,B 0,C 180,E1 -13901.123,E2 -13901.123} C_VEL
LIN {X 0,Y 350.295,Z 247.583,A -85,B 0,C 180,E1 -13901.554,E2 -13901.554} C_VEL
LIN {X 0,Y 354.828,Z 259.276,A -85,B 0,C 180,E1 -13902.172,E2 -13902.172} C_VEL
LIN {X 0,Y 358.206,Z 276.359,A -85,B 0,C 180,E1 -13902.807,E2 -13902.807} C_VEL
LIN {X 0,Y 356.341,Z 355.973,A -85,B 0,C 180,E1 -13904.487,E2 -13904.487} C_VEL
LIN {X 0,Y 355.682,Z 369.801,A -85,B 0,C 180,E1 -13905.03,E2 -13905.03} C_VEL
LIN {X 0,Y 354.883,Z 381.749,A -85,B 0,C 180,E1 -13905.721,E2 -13905.721} C_VEL
LIN {X 0,Y 353.958,Z 392.703,A -85,B 0,C 180,E1 -13906.568,E2 -13906.568} C_VEL
LIN {X 0,Y 352.889,Z 402.879,A -85,B 0,C 180,E1 -13907.559,E2 -13907.559} C_VEL
LIN {X 0,Y 351.754,Z 412.75,A -85,B 0,C 180,E1 -13908.751,E2 -13908.751} C_VEL
LIN {X 0,Y 350.447,Z 422.887,A -85,B 0,C 180,E1 -13910.265,E2 -13910.265} C_VEL
LIN {X 0,Y 349.343,Z 431.583,A -85,B 0,C 180,E1 -13911.896,E2 -13911.896} C_VEL
LIN {X 0,Y 348.208,Z 439.811,A -85,B 0,C 180,E1 -13913.837,E2 -13913.837} C_VEL
LIN {X 0,Y 347.517,Z 445.418,A -85,B 0,C 180,E1 -13915.51,E2 -13915.51} C_VEL
LIN {X 0,Y 346.919,Z 450.684,A -85,B 0,C 180,E1 -13917.531,E2 -13917.531} C_VEL
LIN {X 0,Y 346.464,Z 454.446,A -85,B 0,C 180,E1 -13919.528,E2 -13919.528} C_VEL
LIN {X 0,Y 346.245,Z 456.241,A -85,B 0,C 180,E1 -13920.847,E2 -13920.847} C_VEL
LIN {X 0,Y 346.055,Z 457.488,A -85,B 0,C 180,E1 -13922.153,E2 -13922.153} C_VEL
LIN {X 0,Y 345.963,Z 458.212,A -85,B 0,C 180,E1 -13923.454,E2 -13923.454} C_VEL
LIN {X 0,Y 345.901,Z 458.476,A -85,B 0,C 180,E1 -13924.743,E2 -13924.743} C_VEL
LIN {X 0,Y 345.857,Z 458.169,A -85,B 0,C 180,E1 -13926.125,E2 -13926.125} C_VEL
LIN {X 0,Y 345.91,Z 457.496,A -85,B 0,C 180,E1 -13927.292,E2 -13927.292} C_VEL
LIN {X 0,Y 346.131,Z 455.679,A -85,B 0,C 180,E1 -13929.069,E2 -13929.069} C_VEL
LIN {X 0,Y 346.518,Z 452.478,A -85,B 0,C 180,E1 -13931.064,E2 -13931.064} C_VEL
LIN {X 0,Y 346.856,Z 448.311,A -85,B 0,C 180,E1 -13932.914,E2 -13932.914} C_VEL
LIN {X 0,Y 347.402,Z 442.867,A -85,B 0,C 180,E1 -13934.752,E2 -13934.752} C_VEL
LIN {X 0,Y 348.207,Z 435.955,A -85,B 0,C 180,E1 -13936.579,E2 -13936.579} C_VEL
LIN {X 0,Y 349.184,Z 427.361,A -85,B 0,C 180,E1 -13938.389,E2 -13938.389} C_VEL
LIN {X 0,Y 350.273,Z 417.565,A -85,B 0,C 180,E1 -13940.02,E2 -13940.02} C_VEL
LIN {X 0,Y 351.392,Z 407.439,A -85,B 0,C 180,E1 -13941.373,E2 -13941.373} C_VEL
LIN {X 0,Y 352.492,Z 396.408,A -85,B 0,C 180,E1 -13942.554,E2 -13942.554} C_VEL
LIN {X 0,Y 353.416,Z 384.607,A -85,B 0,C 180,E1 -13943.537,E2 -13943.537} C_VEL
LIN {X 0,Y 354.171,Z 372.423,A -85,B 0,C 180,E1 -13944.306,E2 -13944.306} C_VEL
LIN {X 0,Y 354.85,Z 359.169,A -85,B 0,C 180,E1 -13944.887,E2 -13944.887} C_VEL
LIN {X 0,Y 355.256,Z 343.436,A -85,B 0,C 180,E1 -13945.284,E2 -13945.284} C_VEL
LIN {X 0,Y 356.59,Z 275.08,A -85,B 0,C 180,E1 -13946.688,E2 -13946.688} C_VEL
LIN {X 0,Y 352.538,Z 254.608,A -85,B 0,C 180,E1 -13947.383,E2 -13947.383} C_VEL
LIN {X 0,Y 350.158,Z 247.382,A -85,B 0,C 180,E1 -13947.699,E2 -13947.699} C_VEL
LIN {X 0,Y 348.123,Z 236.124,A -85,B 0,C 180,E1 -13950.976,E2 -13950.976} C_VEL
LIN {X 0,Y 348.192,Z 236.114,A -85,B 0,C 180,E1 -13952.313,E2 -13952.313} C_VEL
LIN {X 0,Y 348.057,Z 236.126,A -85,B 0,C 180,E1 -13956.958,E2 -13956.958} C_VEL
LIN {X 0,Y 347.899,Z 236.146,A -85,B 0,C 180,E1 -13960.475,E2 -13960.475} C_VEL
LIN {X 0,Y 347.901,Z 236.148,A -85,B 0,C 180,E1 -13964.149,E2 -13964.149} C_VEL
LIN {X 0,Y 347.893,Z 236.148,A -85,B 0,C 180,E1 -13968.29,E2 -13968.29} C_VEL
LIN {X 0,Y 347.851,Z 236.151,A -85,B 0,C 180,E1 -13968.873,E2 -13968.873} C_VEL
LIN {X 0,Y 347.111,Z 236.25,A -85,B 0,C 180,E1 -13969.838,E2 -13969.838} C_VEL
LIN {X 0,Y 344.198,Z 236.609,A -85,B 0,C 180,E1 -13971.408,E2 -13971.408} C_VEL
LIN {X 0,Y 341.79,Z 236.906,A -85,B 0,C 180,E1 -13972.679,E2 -13972.679} C_VEL
LIN {X 0,Y 340.794,Z 237.035,A -85,B 0,C 180,E1 -13973.664,E2 -13973.664} C_VEL
LIN {X 0,Y 340.73,Z 237.038,A -85,B 0,C 180,E1 -13973.997,E2 -13973.997} C_VEL
LIN {X 0,Y 340.703,Z 237.044,A -85,B 0,C 180,E1 -13977.5,E2 -13977.5} C_VEL
LIN {X 0,Y 340.695,Z 237.043,A -85,B 0,C 180,E1 -13981.044,E2 -13981.044} C_VEL
LIN {X 0,Y 340.718,Z 237.041,A -85,B 0,C 180,E1 -13985.278,E2 -13985.278} C_VEL
LIN {X 0,Y 340.708,Z 237.043,A -85,B 0,C 180,E1 -13988.385,E2 -13988.385} C_VEL
LIN {X 0,Y 340.697,Z 237.048,A -85,B 0,C 180,E1 -13992.045,E2 -13992.045} C_VEL
LIN {X 0,Y 340.651,Z 237.052,A -85,B 0,C 180,E1 -13996.226,E2 -13996.226} C_VEL
LIN {X 0,Y 340.687,Z 237.048,A -85,B 0,C 180,E1 -13999.752,E2 -13999.752} C_VEL
LIN {X 0,Y 340.703,Z 237.042,A -85,B 0,C 180,E1 -14003.258,E2 -14003.258} C_VEL
LIN {X 0,Y 340.691,Z 237.048,A -85,B 0,C 180,E1 -14006.153,E2 -14006.153} C_VEL
LIN {X 0,Y 340.74,Z 237.041,A -85,B 0,C 180,E1 -14010.329,E2 -14010.329} C_VEL
LIN {X 0,Y 340.801,Z 237.029,A -85,B 0,C 180,E1 -14013.02,E2 -14013.02} C_VEL
LIN {X 0,Y 340.727,Z 237.038,A -85,B 0,C 180,E1 -14016.927,E2 -14016.927} C_VEL
LIN {X 0,Y 340.79,Z 237.032,A -85,B 0,C 180,E1 -14020.733,E2 -14020.733} C_VEL
LIN {X 0,Y 340.784,Z 237.032,A -85,B 0,C 180,E1 -14023.218,E2 -14023.218} C_VEL
LIN {X 0,Y 340.842,Z 237.024,A -85,B 0,C 180,E1 -14026.89,E2 -14026.89} C_VEL
LIN {X 0,Y 340.926,Z 237.016,A -85,B 0,C 180,E1 -14030.508,E2 -14030.508} C_VEL
LIN {X 0,Y 341.073,Z 236.996,A -85,B 0,C 180,E1 -14032.898,E2 -14032.898} C_VEL
LIN {X 0,Y 341.167,Z 236.985,A -85,B 0,C 180,E1 -14037.639,E2 -14037.639} C_VEL
LIN {X 0,Y 341.292,Z 236.973,A -85,B 0,C 180,E1 -14040,E2 -14040} C_VEL
LIN {X 0,Y 341.167,Z 236.988,A -85,B 0,C 180,E1 -14042.361,E2 -14042.361} C_VEL
LIN {X 0,Y 341.073,Z 236.996,A -85,B 0,C 180,E1 -14047.102,E2 -14047.102} C_VEL
LIN {X 0,Y 340.868,Z 237.023,A -85,B 0,C 180,E1 -14050.694,E2 -14050.694} C_VEL
LIN {X 0,Y 340.86,Z 237.028,A -85,B 0,C 180,E1 -14054.325,E2 -14054.325} C_VEL
LIN {X 0,Y 340.835,Z 237.03,A -85,B 0,C 180,E1 -14058.467,E2 -14058.467} C_VEL
LIN {X 0,Y 340.751,Z 237.038,A -85,B 0,C 180,E1 -14061.857,E2 -14061.857} C_VEL
LIN {X 0,Y 340.771,Z 237.034,A -85,B 0,C 180,E1 -14065.665,E2 -14065.665} C_VEL
LIN {X 0,Y 340.739,Z 237.044,A -85,B 0,C 180,E1 -14068.32,E2 -14068.32} C_VEL
LIN {X 0,Y 340.701,Z 237.043,A -85,B 0,C 180,E1 -14071.044,E2 -14071.044} C_VEL
LIN {X 0,Y 340.716,Z 237.04,A -85,B 0,C 180,E1 -14075.279,E2 -14075.279} C_VEL
LIN {X 0,Y 340.708,Z 237.048,A -85,B 0,C 180,E1 -14078.386,E2 -14078.386} C_VEL
LIN {X 0,Y 340.697,Z 237.045,A -85,B 0,C 180,E1 -14082.046,E2 -14082.046} C_VEL
LIN {X 0,Y 340.651,Z 237.053,A -85,B 0,C 180,E1 -14086.227,E2 -14086.227} C_VEL
LIN {X 0,Y 340.687,Z 237.045,A -85,B 0,C 180,E1 -14089.753,E2 -14089.753} C_VEL
LIN {X 0,Y 340.706,Z 237.042,A -85,B 0,C 180,E1 -14093.259,E2 -14093.259} C_VEL
LIN {X 0,Y 340.692,Z 237.047,A -85,B 0,C 180,E1 -14096.154,E2 -14096.154} C_VEL
LIN {X 0,Y 340.746,Z 237.057,A -85,B 0,C 180,E1 -14099.449,E2 -14099.449} C_VEL
LIN {X 0,Y 343.153,Z 248.167,A -85,B 0,C 180,E1 -14102.561,E2 -14102.561} C_VEL
LIN {X 0,Y 344.647,Z 257.168,A -85,B 0,C 180,E1 -14104.968,E2 -14104.968} C_VEL
LIN {X 0,Y 343.872,Z 265.099,A -85,B 0,C 180,E1 -14106.917,E2 -14106.917} C_VEL
LIN {X 0,Y 349.517,Z 300.41,A -85,B 0,C 180,E1 -14108.081,E2 -14108.081} C_VEL
LIN {X 0,Y 348.075,Z 373.898,A -85,B 0,C 180,E1 -14109.656,E2 -14109.656} C_VEL
LIN {X 0,Y 347.398,Z 386.887,A -85,B 0,C 180,E1 -14110.154,E2 -14110.154} C_VEL
LIN {X 0,Y 346.389,Z 400.037,A -85,B 0,C 180,E1 -14110.904,E2 -14110.904} C_VEL
LIN {X 0,Y 345.268,Z 412.725,A -85,B 0,C 180,E1 -14111.916,E2 -14111.916} C_VEL
LIN {X 0,Y 344.093,Z 424.022,A -85,B 0,C 180,E1 -14113.079,E2 -14113.079} C_VEL
LIN {X 0,Y 343.025,Z 433.898,A -85,B 0,C 180,E1 -14114.355,E2 -14114.355} C_VEL
LIN {X 0,Y 342.049,Z 442.547,A -85,B 0,C 180,E1 -14115.726,E2 -14115.726} C_VEL
LIN {X 0,Y 341.143,Z 450.255,A -85,B 0,C 180,E1 -14117.205,E2 -14117.205} C_VEL
LIN {X 0,Y 340.269,Z 457.799,A -85,B 0,C 180,E1 -14118.986,E2 -14118.986} C_VEL
LIN {X 0,Y 339.614,Z 464.765,A -85,B 0,C 180,E1 -14121.072,E2 -14121.072} C_VEL
LIN {X 0,Y 339.27,Z 469.351,A -85,B 0,C 180,E1 -14122.86,E2 -14122.86} C_VEL
LIN {X 0,Y 339.132,Z 471.874,A -85,B 0,C 180,E1 -14124.115,E2 -14124.115} C_VEL
LIN {X 0,Y 339.07,Z 475.291,A -85,B 0,C 180,E1 -14126.435,E2 -14126.435} C_VEL
LIN {X 0,Y 338.999,Z 476.392,A -85,B 0,C 180,E1 -14127.624,E2 -14127.624} C_VEL
LIN {X 0,Y 339.019,Z 477.081,A -85,B 0,C 180,E1 -14128.812,E2 -14128.812} C_VEL
LIN {X 0,Y 339.067,Z 477.38,A -85,B 0,C 180,E1 -14130,E2 -14130} C_VEL
LIN {X 0,Y 339.005,Z 477.287,A -85,B 0,C 180,E1 -14131.188,E2 -14131.188} C_VEL
LIN {X 0,Y 338.997,Z 476.767,A -85,B 0,C 180,E1 -14132.377,E2 -14132.377} C_VEL
LIN {X 0,Y 339.065,Z 475.836,A -85,B 0,C 180,E1 -14133.565,E2 -14133.565} C_VEL
LIN {X 0,Y 339.111,Z 472.923,A -85,B 0,C 180,E1 -14135.85,E2 -14135.85} C_VEL
LIN {X 0,Y 339.397,Z 469.294,A -85,B 0,C 180,E1 -14137.735,E2 -14137.735} C_VEL
LIN {X 0,Y 339.823,Z 464.735,A -85,B 0,C 180,E1 -14139.524,E2 -14139.524} C_VEL
LIN {X 0,Y 340.6,Z 457.839,A -85,B 0,C 180,E1 -14141.606,E2 -14141.606} C_VEL
LIN {X 0,Y 341.703,Z 450.37,A -85,B 0,C 180,E1 -14143.379,E2 -14143.379} C_VEL
LIN {X 0,Y 342.692,Z 442.77,A -85,B 0,C 180,E1 -14144.854,E2 -14144.854} C_VEL
LIN {X 0,Y 343.933,Z 432.756,A -85,B 0,C 180,E1 -14146.439,E2 -14146.439} C_VEL
LIN {X 0,Y 345.285,Z 422.103,A -85,B 0,C 180,E1 -14147.777,E2 -14147.777} C_VEL
LIN {X 0,Y 346.674,Z 410.545,A -85,B 0,C 180,E1 -14148.927,E2 -14148.927} C_VEL
LIN {X 0,Y 347.824,Z 399.463,A -85,B 0,C 180,E1 -14149.782,E2 -14149.782} C_VEL
LIN {X 0,Y 348.856,Z 386.359,A -85,B 0,C 180,E1 -14150.528,E2 -14150.528} C_VEL
LIN {X 0,Y 349.649,Z 373.466,A -85,B 0,C 180,E1 -14151.018,E2 -14151.018} C_VEL
LIN {X 0,Y 351.129,Z 300.8,A -85,B 0,C 180,E1 -14152.598,E2 -14152.598} C_VEL
LIN {X 0,Y 347.411,Z 277.908,A -85,B 0,C 180,E1 -14153.407,E2 -14153.407} C_VEL
LIN {X 0,Y 344.653,Z 264.272,A -85,B 0,C 180,E1 -14153.953,E2 -14153.953} C_VEL
LIN {X 0,Y 345.193,Z 258.704,A -85,B 0,C 180,E1 -14155.312,E2 -14155.312} C_VEL
LIN {X 0,Y 343.236,Z 247.689,A -85,B 0,C 180,E1 -14158.302,E2 -14158.302} C_VEL
LIN {X 0,Y 340.729,Z 237.046,A -85,B 0,C 180,E1 -14161.387,E2 -14161.387} C_VEL
LIN {X 0,Y 340.719,Z 237.048,A -85,B 0,C 180,E1 -14165.279,E2 -14165.279} C_VEL
LIN {X 0,Y 340.71,Z 237.043,A -85,B 0,C 180,E1 -14168.386,E2 -14168.386} C_VEL
LIN {X 0,Y 340.7,Z 237.044,A -85,B 0,C 180,E1 -14172.045,E2 -14172.045} C_VEL
LIN {X 0,Y 340.652,Z 237.052,A -85,B 0,C 180,E1 -14176.227,E2 -14176.227} C_VEL
LIN {X 0,Y 340.688,Z 237.048,A -85,B 0,C 180,E1 -14179.753,E2 -14179.753} C_VEL
LIN {X 0,Y 340.705,Z 237.047,A -85,B 0,C 180,E1 -14183.258,E2 -14183.258} C_VEL
LIN {X 0,Y 340.692,Z 237.044,A -85,B 0,C 180,E1 -14186.153,E2 -14186.153} C_VEL
LIN {X 0,Y 340.741,Z 237.038,A -85,B 0,C 180,E1 -14190.329,E2 -14190.329} C_VEL
LIN {X 0,Y 340.803,Z 237.026,A -85,B 0,C 180,E1 -14193.02,E2 -14193.02} C_VEL
LIN {X 0,Y 340.756,Z 237.035,A -85,B 0,C 180,E1 -14195.638,E2 -14195.638} C_VEL
LIN {X 0,Y 340.748,Z 237.039,A -85,B 0,C 180,E1 -14199.474,E2 -14199.474} C_VEL
LIN {X 0,Y 340.858,Z 237.019,A -85,B 0,C 180,E1 -14201.984,E2 -14201.984} C_VEL
LIN {X 0,Y 340.869,Z 237.013,A -85,B 0,C 180,E1 -14205.705,E2 -14205.705} C_VEL
LIN {X 0,Y 340.87,Z 237.019,A -85,B 0,C 180,E1 -14209.306,E2 -14209.306} C_VEL
LIN {X 0,Y 341.059,Z 237.003,A -85,B 0,C 180,E1 -14212.898,E2 -14212.898} C_VEL
LIN {X 0,Y 341.169,Z 236.986,A -85,B 0,C 180,E1 -14217.639,E2 -14217.639} C_VEL
LIN {X 0,Y 341.275,Z 236.964,A -85,B 0,C 180,E1 -14220,E2 -14220} C_VEL
LIN {X 0,Y 341.168,Z 236.988,A -85,B 0,C 180,E1 -14222.361,E2 -14222.361} C_VEL
LIN {X 0,Y 341.074,Z 236.995,A -85,B 0,C 180,E1 -14227.102,E2 -14227.102} C_VEL
LIN {X 0,Y 340.87,Z 237.024,A -85,B 0,C 180,E1 -14230.694,E2 -14230.694} C_VEL
LIN {X 0,Y 340.863,Z 237.027,A -85,B 0,C 180,E1 -14234.325,E2 -14234.325} C_VEL
LIN {X 0,Y 340.838,Z 237.026,A -85,B 0,C 180,E1 -14238.467,E2 -14238.467} C_VEL
LIN {X 0,Y 340.717,Z 237.042,A -85,B 0,C 180,E1 -14241.842,E2 -14241.842} C_VEL
LIN {X 0,Y 340.745,Z 237.04,A -85,B 0,C 180,E1 -14245.667,E2 -14245.667} C_VEL
LIN {X 0,Y 340.732,Z 237.036,A -85,B 0,C 180,E1 -14249.672,E2 -14249.672} C_VEL
LIN {X 0,Y 340.692,Z 237.052,A -85,B 0,C 180,E1 -14253.847,E2 -14253.847} C_VEL
LIN {X 0,Y 340.74,Z 237.044,A -85,B 0,C 180,E1 -14257.758,E2 -14257.758} C_VEL
LIN {X 0,Y 343.127,Z 247.691,A -85,B 0,C 180,E1 -14260.953,E2 -14260.953} C_VEL
LIN {X 0,Y 348.676,Z 261.849,A -85,B 0,C 180,E1 -14261.758,E2 -14261.758} C_VEL
LIN {X 0,Y 351.689,Z 276.444,A -85,B 0,C 180,E1 -14262.326,E2 -14262.326} C_VEL
LIN {X 0,Y 349.852,Z 355.106,A -85,B 0,C 180,E1 -14264.011,E2 -14264.011} C_VEL
LIN {X 0,Y 349.204,Z 368.198,A -85,B 0,C 180,E1 -14264.509,E2 -14264.509} C_VEL
LIN {X 0,Y 348.305,Z 381.575,A -85,B 0,C 180,E1 -14265.276,E2 -14265.276} C_VEL
LIN {X 0,Y 347.338,Z 392.555,A -85,B 0,C 180,E1 -14266.131,E2 -14266.131} C_VEL
LIN {X 0,Y 346.138,Z 403.606,A -85,B 0,C 180,E1 -14267.233,E2 -14267.233} C_VEL
LIN {X 0,Y 344.912,Z 413.66,A -85,B 0,C 180,E1 -14268.486,E2 -14268.486} C_VEL
LIN {X 0,Y 343.654,Z 422.858,A -85,B 0,C 180,E1 -14269.894,E2 -14269.894} C_VEL
LIN {X 0,Y 342.443,Z 431.73,A -85,B 0,C 180,E1 -14271.581,E2 -14271.581} C_VEL
LIN {X 0,Y 341.368,Z 439.401,A -85,B 0,C 180,E1 -14273.411,E2 -14273.411} C_VEL
LIN {X 0,Y 340.515,Z 445.546,A -85,B 0,C 180,E1 -14275.254,E2 -14275.254} C_VEL
LIN {X 0,Y 339.849,Z 451.161,A -85,B 0,C 180,E1 -14277.475,E2 -14277.475} C_VEL
LIN {X 0,Y 339.375,Z 454.843,A -85,B 0,C 180,E1 -14279.512,E2 -14279.512} C_VEL
LIN {X 0,Y 339.03,Z 457.24,A -85,B 0,C 180,E1 -14281.524,E2 -14281.524} C_VEL
LIN {X 0,Y 338.887,Z 458.297,A -85,B 0,C 180,E1 -14283.095,E2 -14283.095} C_VEL
LIN {X 0,Y 338.784,Z 458.571,A -85,B 0,C 180,E1 -14285.487,E2 -14285.487} C_VEL
LIN {X 0,Y 338.779,Z 458.048,A -85,B 0,C 180,E1 -14286.787,E2 -14286.787} C_VEL
LIN {X 0,Y 339.002,Z 456.151,A -85,B 0,C 180,E1 -14288.895,E2 -14288.895} C_VEL
LIN {X 0,Y 339.462,Z 452.439,A -85,B 0,C 180,E1 -14291.282,E2 -14291.282} C_VEL
LIN {X 0,Y 339.836,Z 448.176,A -85,B 0,C 180,E1 -14293.17,E2 -14293.17} C_VEL
LIN {X 0,Y 340.565,Z 441.561,A -85,B 0,C 180,E1 -14295.357,E2 -14295.357} C_VEL
LIN {X 0,Y 341.419,Z 434.33,A -85,B 0,C 180,E1 -14297.215,E2 -14297.215} C_VEL
LIN {X 0,Y 342.319,Z 426.892,A -85,B 0,C 180,E1 -14298.753,E2 -14298.753} C_VEL
LIN {X 0,Y 343.428,Z 417.416,A -85,B 0,C 180,E1 -14300.341,E2 -14300.341} C_VEL
LIN {X 0,Y 344.574,Z 406.664,A -85,B 0,C 180,E1 -14301.792,E2 -14301.792} C_VEL
LIN {X 0,Y 345.798,Z 395.257,A -85,B 0,C 180,E1 -14302.996,E2 -14302.996} C_VEL
LIN {X 0,Y 346.743,Z 383.595,A -85,B 0,C 180,E1 -14303.96,E2 -14303.96} C_VEL
LIN {X 0,Y 347.462,Z 371.753,A -85,B 0,C 180,E1 -14304.705,E2 -14304.705} C_VEL
LIN {X 0,Y 348.129,Z 359.013,A -85,B 0,C 180,E1 -14305.259,E2 -14305.259} C_VEL
LIN {X 0,Y 348.552,Z 343.354,A -85,B 0,C 180,E1 -14305.658,E2 -14305.658} C_VEL
LIN {X 0,Y 349.851,Z 275.407,A -85,B 0,C 180,E1 -14307.086,E2 -14307.086} C_VEL
LIN {X 0,Y 346.023,Z 256.448,A -85,B 0,C 180,E1 -14307.752,E2 -14307.752} C_VEL
LIN {X 0,Y 343.071,Z 247.491,A -85,B 0,C 180,E1 -14308.177,E2 -14308.177} C_VEL
LIN {X 0,Y 341.076,Z 237.001,A -85,B 0,C 180,E1 -14311.328,E2 -14311.328} C_VEL
LIN {X 0,Y 341.129,Z 236.995,A -85,B 0,C 180,E1 -14312.361,E2 -14312.361} C_VEL
LIN {X 0,Y 341.018,Z 237.008,A -85,B 0,C 180,E1 -14315.914,E2 -14315.914} C_VEL
LIN {X 0,Y 340.966,Z 237.011,A -85,B 0,C 180,E1 -14318.356,E2 -14318.356} C_VEL
LIN {X 0,Y 340.852,Z 237.029,A -85,B 0,C 180,E1 -14321.899,E2 -14321.899} C_VEL
LIN {X 0,Y 340.821,Z 237.031,A -85,B 0,C 180,E1 -14325.549,E2 -14325.549} C_VEL
LIN {X 0,Y 340.807,Z 237.029,A -85,B 0,C 180,E1 -14328.861,E2 -14328.861} C_VEL
LIN {X 0,Y 340.722,Z 237.039,A -85,B 0,C 180,E1 -14333.073,E2 -14333.073} C_VEL
LIN {X 0,Y 340.73,Z 237.038,A -85,B 0,C 180,E1 -14333.997,E2 -14333.997} C_VEL
LIN {X 0,Y 340.106,Z 237.119,A -85,B 0,C 180,E1 -14334.983,E2 -14334.983} C_VEL
LIN {X 0,Y 337.257,Z 237.476,A -85,B 0,C 180,E1 -14336.587,E2 -14336.587} C_VEL
LIN {X 0,Y 334.805,Z 237.782,A -85,B 0,C 180,E1 -14337.886,E2 -14337.886} C_VEL
LIN {X 0,Y 333.737,Z 237.909,A -85,B 0,C 180,E1 -14338.891,E2 -14338.891} C_VEL
LIN {X 0,Y 333.644,Z 237.92,A -85,B 0,C 180,E1 -14339.232,E2 -14339.232} C_VEL
LIN {X 0,Y 333.637,Z 237.923,A -85,B 0,C 180,E1 -14343.208,E2 -14343.208} C_VEL
LIN {X 0,Y 333.676,Z 237.921,A -85,B 0,C 180,E1 -14346.138,E2 -14346.138} C_VEL
LIN {X 0,Y 333.646,Z 237.922,A -85,B 0,C 180,E1 -14349.192,E2 -14349.192} C_VEL
LIN {X 0,Y 333.631,Z 237.923,A -85,B 0,C 180,E1 -14352.499,E2 -14352.499} C_VEL
LIN {X 0,Y 333.596,Z 237.932,A -85,B 0,C 180,E1 -14355.955,E2 -14355.955} C_VEL
LIN {X 0,Y 333.646,Z 237.922,A -85,B 0,C 180,E1 -14359.315,E2 -14359.315} C_VEL
LIN {X 0,Y 333.664,Z 237.918,A -85,B 0,C 180,E1 -14363.167,E2 -14363.167} C_VEL
LIN {X 0,Y 333.673,Z 237.917,A -85,B 0,C 180,E1 -14365.341,E2 -14365.341} C_VEL
LIN {X 0,Y 333.689,Z 237.918,A -85,B 0,C 180,E1 -14369.637,E2 -14369.637} C_VEL
LIN {X 0,Y 333.738,Z 237.912,A -85,B 0,C 180,E1 -14372.4,E2 -14372.4} C_VEL
LIN {X 0,Y 333.725,Z 237.909,A -85,B 0,C 180,E1 -14375.09,E2 -14375.09} C_VEL
LIN {X 0,Y 333.678,Z 237.916,A -85,B 0,C 180,E1 -14379.019,E2 -14379.019} C_VEL
LIN {X 0,Y 333.792,Z 237.904,A -85,B 0,C 180,E1 -14381.589,E2 -14381.589} C_VEL
LIN {X 0,Y 333.806,Z 237.902,A -85,B 0,C 180,E1 -14385.576,E2 -14385.576} C_VEL
LIN {X 0,Y 333.831,Z 237.895,A -85,B 0,C 180,E1 -14389.078,E2 -14389.078} C_VEL
LIN {X 0,Y 334.023,Z 237.875,A -85,B 0,C 180,E1 -14392.747,E2 -14392.747} C_VEL
LIN {X 0,Y 333.808,Z 237.901,A -85,B 0,C 180,E1 -14395.169,E2 -14395.169} C_VEL
LIN {X 0,Y 334.105,Z 237.865,A -85,B 0,C 180,E1 -14397.589,E2 -14397.589} C_VEL
LIN {X 0,Y 334.243,Z 237.85,A -85,B 0,C 180,E1 -14400,E2 -14400} C_VEL
LIN {X 0,Y 334.105,Z 237.866,A -85,B 0,C 180,E1 -14402.411,E2 -14402.411} C_VEL
LIN {X 0,Y 334.023,Z 237.874,A -85,B 0,C 180,E1 -14407.252,E2 -14407.252} C_VEL
LIN {X 0,Y 333.831,Z 237.898,A -85,B 0,C 180,E1 -14410.922,E2 -14410.922} C_VEL
LIN {X 0,Y 333.806,Z 237.903,A -85,B 0,C 180,E1 -14414.634,E2 -14414.634} C_VEL
LIN {X 0,Y 333.795,Z 237.905,A -85,B 0,C 180,E1 -14418.656,E2 -14418.656} C_VEL
LIN {X 0,Y 333.69,Z 237.921,A -85,B 0,C 180,E1 -14422.278,E2 -14422.278} C_VEL
LIN {X 0,Y 333.734,Z 237.916,A -85,B 0,C 180,E1 -14426.246,E2 -14426.246} C_VEL
LIN {X 0,Y 333.709,Z 237.914,A -85,B 0,C 180,E1 -14428.972,E2 -14428.972} C_VEL
LIN {X 0,Y 333.641,Z 237.925,A -85,B 0,C 180,E1 -14432.587,E2 -14432.587} C_VEL
LIN {X 0,Y 333.674,Z 237.922,A -85,B 0,C 180,E1 -14436.139,E2 -14436.139} C_VEL
LIN {X 0,Y 333.645,Z 237.922,A -85,B 0,C 180,E1 -14439.193,E2 -14439.193} C_VEL
LIN {X 0,Y 333.631,Z 237.927,A -85,B 0,C 180,E1 -14442.5,E2 -14442.5} C_VEL
LIN {X 0,Y 333.595,Z 237.93,A -85,B 0,C 180,E1 -14445.955,E2 -14445.955} C_VEL
LIN {X 0,Y 333.646,Z 237.921,A -85,B 0,C 180,E1 -14449.316,E2 -14449.316} C_VEL
LIN {X 0,Y 333.666,Z 237.92,A -85,B 0,C 180,E1 -14453.168,E2 -14453.168} C_VEL
LIN {X 0,Y 333.636,Z 237.928,A -85,B 0,C 180,E1 -14456.792,E2 -14456.792} C_VEL
LIN {X 0,Y 333.715,Z 238.033,A -85,B 0,C 180,E1 -14459.115,E2 -14459.115} C_VEL
LIN {X 0,Y 335.983,Z 248.487,A -85,B 0,C 180,E1 -14462.115,E2 -14462.115} C_VEL
LIN {X 0,Y 337.671,Z 258.072,A -85,B 0,C 180,E1 -14464.744,E2 -14464.744} C_VEL
LIN {X 0,Y 337.079,Z 264.972,A -85,B 0,C 180,E1 -14466.484,E2 -14466.484} C_VEL
LIN {X 0,Y 342.918,Z 301.942,A -85,B 0,C 180,E1 -14467.714,E2 -14467.714} C_VEL
LIN {X 0,Y 341.36,Z 373.682,A -85,B 0,C 180,E1 -14469.277,E2 -14469.277} C_VEL
LIN {X 0,Y 340.669,Z 386.675,A -85,B 0,C 180,E1 -14469.785,E2 -14469.785} C_VEL
LIN {X 0,Y 339.652,Z 399.284,A -85,B 0,C 180,E1 -14470.51,E2 -14470.51} C_VEL
LIN {X 0,Y 338.686,Z 410.538,A -85,B 0,C 180,E1 -14471.395,E2 -14471.395} C_VEL
LIN {X 0,Y 337.389,Z 422.193,A -85,B 0,C 180,E1 -14472.576,E2 -14472.576} C_VEL
LIN {X 0,Y 336.239,Z 432.701,A -85,B 0,C 180,E1 -14473.923,E2 -14473.923} C_VEL
LIN {X 0,Y 335.146,Z 442.144,A -85,B 0,C 180,E1 -14475.426,E2 -14475.426} C_VEL
LIN {X 0,Y 334.033,Z 451.254,A -85,B 0,C 180,E1 -14477.237,E2 -14477.237} C_VEL
LIN {X 0,Y 333.142,Z 458.59,A -85,B 0,C 180,E1 -14479.055,E2 -14479.055} C_VEL
LIN {X 0,Y 332.571,Z 464.461,A -85,B 0,C 180,E1 -14480.881,E2 -14480.881} C_VEL
LIN {X 0,Y 332.196,Z 469.073,A -85,B 0,C 180,E1 -14482.708,E2 -14482.708} C_VEL
LIN {X 0,Y 332.029,Z 471.947,A -85,B 0,C 180,E1 -14484.179,E2 -14484.179} C_VEL
LIN {X 0,Y 331.995,Z 475.052,A -85,B 0,C 180,E1 -14486.359,E2 -14486.359} C_VEL
LIN {X 0,Y 331.916,Z 476.172,A -85,B 0,C 180,E1 -14487.573,E2 -14487.573} C_VEL
LIN {X 0,Y 331.924,Z 476.87,A -85,B 0,C 180,E1 -14488.787,E2 -14488.787} C_VEL
LIN {X 0,Y 331.969,Z 477.178,A -85,B 0,C 180,E1 -14490,E2 -14490} C_VEL
LIN {X 0,Y 331.912,Z 477.094,A -85,B 0,C 180,E1 -14491.213,E2 -14491.213} C_VEL
LIN {X 0,Y 331.915,Z 476.593,A -85,B 0,C 180,E1 -14492.427,E2 -14492.427} C_VEL
LIN {X 0,Y 331.968,Z 475.67,A -85,B 0,C 180,E1 -14493.642,E2 -14493.642} C_VEL
LIN {X 0,Y 332.006,Z 473.065,A -85,B 0,C 180,E1 -14495.781,E2 -14495.781} C_VEL
LIN {X 0,Y 332.353,Z 469.164,A -85,B 0,C 180,E1 -14497.9,E2 -14497.9} C_VEL
LIN {X 0,Y 332.798,Z 464.624,A -85,B 0,C 180,E1 -14499.727,E2 -14499.727} C_VEL
LIN {X 0,Y 333.616,Z 457.762,A -85,B 0,C 180,E1 -14501.853,E2 -14501.853} C_VEL
LIN {X 0,Y 334.765,Z 450.329,A -85,B 0,C 180,E1 -14503.661,E2 -14503.661} C_VEL
LIN {X 0,Y 336.021,Z 441.106,A -85,B 0,C 180,E1 -14505.466,E2 -14505.466} C_VEL
LIN {X 0,Y 337.292,Z 431.54,A -85,B 0,C 180,E1 -14506.961,E2 -14506.961} C_VEL
LIN {X 0,Y 338.698,Z 420.951,A -85,B 0,C 180,E1 -14508.291,E2 -14508.291} C_VEL
LIN {X 0,Y 340.178,Z 409.13,A -85,B 0,C 180,E1 -14509.459,E2 -14509.459} C_VEL
LIN {X 0,Y 341.378,Z 397.622,A -85,B 0,C 180,E1 -14510.329,E2 -14510.329} C_VEL
LIN {X 0,Y 342.406,Z 384.697,A -85,B 0,C 180,E1 -14511.051,E2 -14511.051} C_VEL
LIN {X 0,Y 343.141,Z 372.207,A -85,B 0,C 180,E1 -14511.515,E2 -14511.515} C_VEL
LIN {X 0,Y 344.729,Z 302.094,A -85,B 0,C 180,E1 -14513.051,E2 -14513.051} C_VEL
LIN {X 0,Y 341.005,Z 279.057,A -85,B 0,C 180,E1 -14513.89,E2 -14513.89} C_VEL
LIN {X 0,Y 338.015,Z 263.985,A -85,B 0,C 180,E1 -14514.525,E2 -14514.525} C_VEL
LIN {X 0,Y 338.293,Z 259.97,A -85,B 0,C 180,E1 -14515.536,E2 -14515.536} C_VEL
LIN {X 0,Y 336.452,Z 249.734,A -85,B 0,C 180,E1 -14518.383,E2 -14518.383} C_VEL
LIN {X 0,Y 333.687,Z 237.924,A -85,B 0,C 180,E1 -14521.912,E2 -14521.912} C_VEL
LIN {X 0,Y 333.686,Z 237.922,A -85,B 0,C 180,E1 -14524.774,E2 -14524.774} C_VEL
LIN {X 0,Y 333.652,Z 237.923,A -85,B 0,C 180,E1 -14527.651,E2 -14527.651} C_VEL
LIN {X 0,Y 333.647,Z 237.923,A -85,B 0,C 180,E1 -14530.767,E2 -14530.767} C_VEL
LIN {X 0,Y 333.594,Z 237.932,A -85,B 0,C 180,E1 -14534.25,E2 -14534.25} C_VEL
LIN {X 0,Y 333.642,Z 237.922,A -85,B 0,C 180,E1 -14537.618,E2 -14537.618} C_VEL
LIN {X 0,Y 333.652,Z 237.92,A -85,B 0,C 180,E1 -14541.202,E2 -14541.202} C_VEL
LIN {X 0,Y 333.676,Z 237.917,A -85,B 0,C 180,E1 -14543.861,E2 -14543.861} C_VEL
LIN {X 0,Y 333.643,Z 237.922,A -85,B 0,C 180,E1 -14547.413,E2 -14547.413} C_VEL
LIN {X 0,Y 333.69,Z 237.92,A -85,B 0,C 180,E1 -14551.026,E2 -14551.026} C_VEL
LIN {X 0,Y 333.735,Z 237.911,A -85,B 0,C 180,E1 -14553.754,E2 -14553.754} C_VEL
LIN {X 0,Y 333.719,Z 237.912,A -85,B 0,C 180,E1 -14557.914,E2 -14557.914} C_VEL
LIN {X 0,Y 333.794,Z 237.898,A -85,B 0,C 180,E1 -14561.589,E2 -14561.589} C_VEL
LIN {X 0,Y 333.808,Z 237.893,A -85,B 0,C 180,E1 -14565.577,E2 -14565.577} C_VEL
LIN {X 0,Y 333.833,Z 237.898,A -85,B 0,C 180,E1 -14569.078,E2 -14569.078} C_VEL
LIN {X 0,Y 334.012,Z 237.88,A -85,B 0,C 180,E1 -14572.747,E2 -14572.747} C_VEL
LIN {X 0,Y 333.808,Z 237.896,A -85,B 0,C 180,E1 -14575.169,E2 -14575.169} C_VEL
LIN {X 0,Y 334.106,Z 237.866,A -85,B 0,C 180,E1 -14577.589,E2 -14577.589} C_VEL
LIN {X 0,Y 334.227,Z 237.842,A -85,B 0,C 180,E1 -14580,E2 -14580} C_VEL
LIN {X 0,Y 334.105,Z 237.868,A -85,B 0,C 180,E1 -14582.411,E2 -14582.411} C_VEL
LIN {X 0,Y 334.024,Z 237.872,A -85,B 0,C 180,E1 -14587.253,E2 -14587.253} C_VEL
LIN {X 0,Y 333.833,Z 237.898,A -85,B 0,C 180,E1 -14590.922,E2 -14590.922} C_VEL
LIN {X 0,Y 333.808,Z 237.902,A -85,B 0,C 180,E1 -14594.634,E2 -14594.634} C_VEL
LIN {X 0,Y 333.797,Z 237.903,A -85,B 0,C 180,E1 -14598.655,E2 -14598.655} C_VEL
LIN {X 0,Y 333.656,Z 237.924,A -85,B 0,C 180,E1 -14602.281,E2 -14602.281} C_VEL
LIN {X 0,Y 333.705,Z 237.918,A -85,B 0,C 180,E1 -14605.096,E2 -14605.096} C_VEL
LIN {X 0,Y 333.67,Z 237.913,A -85,B 0,C 180,E1 -14608.976,E2 -14608.976} C_VEL
LIN {X 0,Y 333.644,Z 237.921,A -85,B 0,C 180,E1 -14612.587,E2 -14612.587} C_VEL
LIN {X 0,Y 333.675,Z 237.928,A -85,B 0,C 180,E1 -14616.139,E2 -14616.139} C_VEL
LIN {X 0,Y 333.702,Z 237.972,A -85,B 0,C 180,E1 -14617.327,E2 -14617.327} C_VEL
LIN {X 0,Y 336,Z 248.085,A -85,B 0,C 180,E1 -14620.373,E2 -14620.373} C_VEL
LIN {X 0,Y 342.567,Z 264.35,A -85,B 0,C 180,E1 -14621.327,E2 -14621.327} C_VEL
LIN {X 0,Y 345.28,Z 277.826,A -85,B 0,C 180,E1 -14621.864,E2 -14621.864} C_VEL
LIN {X 0,Y 343.299,Z 355.963,A -85,B 0,C 180,E1 -14623.572,E2 -14623.572} C_VEL
LIN {X 0,Y 342.588,Z 369.482,A -85,B 0,C 180,E1 -14624.11,E2 -14624.11} C_VEL
LIN {X 0,Y 341.66,Z 382.602,A -85,B 0,C 180,E1 -14624.897,E2 -14624.897} C_VEL
LIN {X 0,Y 340.535,Z 394.486,A -85,B 0,C 180,E1 -14625.871,E2 -14625.871} C_VEL
LIN {X 0,Y 339.204,Z 405.871,A -85,B 0,C 180,E1 -14627.067,E2 -14627.067} C_VEL
LIN {X 0,Y 338.007,Z 415.182,A -85,B 0,C 180,E1 -14628.29,E2 -14628.29} C_VEL
LIN {X 0,Y 336.736,Z 423.903,A -85,B 0,C 180,E1 -14629.684,E2 -14629.684} C_VEL
LIN {X 0,Y 335.46,Z 432.752,A -85,B 0,C 180,E1 -14631.445,E2 -14631.445} C_VEL
LIN {X 0,Y 334.27,Z 440.719,A -85,B 0,C 180,E1 -14633.433,E2 -14633.433} C_VEL
LIN {X 0,Y 333.425,Z 446.608,A -85,B 0,C 180,E1 -14635.312,E2 -14635.312} C_VEL
LIN {X 0,Y 332.712,Z 452.144,A -85,B 0,C 180,E1 -14637.666,E2 -14637.666} C_VEL
LIN {X 0,Y 332.283,Z 455.24,A -85,B 0,C 180,E1 -14639.495,E2 -14639.495} C_VEL
LIN {X 0,Y 332.035,Z 456.94,A -85,B 0,C 180,E1 -14640.868,E2 -14640.868} C_VEL
LIN {X 0,Y 331.82,Z 458.419,A -85,B 0,C 180,E1 -14642.82,E2 -14642.82} C_VEL
LIN {X 0,Y 331.68,Z 458.846,A -85,B 0,C 180,E1 -14644.926,E2 -14644.926} C_VEL
LIN {X 0,Y 331.661,Z 458.499,A -85,B 0,C 180,E1 -14646.258,E2 -14646.258} C_VEL
LIN {X 0,Y 331.754,Z 457.706,A -85,B 0,C 180,E1 -14647.585,E2 -14647.585} C_VEL
LIN {X 0,Y 331.933,Z 456.392,A -85,B 0,C 180,E1 -14648.903,E2 -14648.903} C_VEL
LIN {X 0,Y 332.3,Z 453.547,A -85,B 0,C 180,E1 -14650.864,E2 -14650.864} C_VEL
LIN {X 0,Y 332.646,Z 449.599,A -85,B 0,C 180,E1 -14652.795,E2 -14652.795} C_VEL
LIN {X 0,Y 333.222,Z 444.417,A -85,B 0,C 180,E1 -14654.714,E2 -14654.714} C_VEL
LIN {X 0,Y 334.051,Z 437.85,A -85,B 0,C 180,E1 -14656.619,E2 -14656.619} C_VEL
LIN {X 0,Y 335.059,Z 429.577,A -85,B 0,C 180,E1 -14658.506,E2 -14658.506} C_VEL
LIN {X 0,Y 336.2,Z 420.412,A -85,B 0,C 180,E1 -14660.18,E2 -14660.18} C_VEL
LIN {X 0,Y 337.295,Z 410.717,A -85,B 0,C 180,E1 -14661.613,E2 -14661.613} C_VEL
LIN {X 0,Y 338.462,Z 400.299,A -85,B 0,C 180,E1 -14662.843,E2 -14662.843} C_VEL
LIN {X 0,Y 339.584,Z 388.593,A -85,B 0,C 180,E1 -14663.938,E2 -14663.938} C_VEL
LIN {X 0,Y 340.482,Z 376.332,A -85,B 0,C 180,E1 -14664.819,E2 -14664.819} C_VEL
LIN {X 0,Y 341.175,Z 363.788,A -85,B 0,C 180,E1 -14665.458,E2 -14665.458} C_VEL
LIN {X 0,Y 341.641,Z 351.283,A -85,B 0,C 180,E1 -14665.871,E2 -14665.871} C_VEL
LIN {X 0,Y 343.187,Z 276.365,A -85,B 0,C 180,E1 -14667.481,E2 -14667.481} C_VEL
LIN {X 0,Y 339.602,Z 258.6,A -85,B 0,C 180,E1 -14668.121,E2 -14668.121} C_VEL
LIN {X 0,Y 335.911,Z 247.758,A -85,B 0,C 180,E1 -14668.633,E2 -14668.633} C_VEL
LIN {X 0,Y 334.05,Z 237.877,A -85,B 0,C 180,E1 -14671.658,E2 -14671.658} C_VEL
LIN {X 0,Y 333.992,Z 237.882,A -85,B 0,C 180,E1 -14676.039,E2 -14676.039} C_VEL
LIN {X 0,Y 333.823,Z 237.905,A -85,B 0,C 180,E1 -14679.696,E2 -14679.696} C_VEL
LIN {X 0,Y 333.799,Z 237.905,A -85,B 0,C 180,E1 -14683.391,E2 -14683.391} C_VEL
LIN {X 0,Y 333.748,Z 237.91,A -85,B 0,C 180,E1 -14687.146,E2 -14687.146} C_VEL
LIN {X 0,Y 333.734,Z 237.915,A -85,B 0,C 180,E1 -14689.69,E2 -14689.69} C_VEL
LIN {X 0,Y 333.671,Z 237.921,A -85,B 0,C 180,E1 -14693.59,E2 -14693.59} C_VEL
LIN {X 0,Y 333.669,Z 237.921,A -85,B 0,C 180,E1 -14696.251,E2 -14696.251} C_VEL
LIN {X 0,Y 333.644,Z 237.92,A -85,B 0,C 180,E1 -14699.232,E2 -14699.232} C_VEL
LIN {X 0,Y 332.958,Z 238.01,A -85,B 0,C 180,E1 -14700.241,E2 -14700.241} C_VEL
LIN {X 0,Y 330.098,Z 238.369,A -85,B 0,C 180,E1 -14701.881,E2 -14701.881} C_VEL
LIN {X 0,Y 327.694,Z 238.667,A -85,B 0,C 180,E1 -14703.21,E2 -14703.21} C_VEL
LIN {X 0,Y 326.675,Z 238.792,A -85,B 0,C 180,E1 -14704.239,E2 -14704.239} C_VEL
LIN {X 0,Y 326.598,Z 238.798,A -85,B 0,C 180,E1 -14704.587,E2 -14704.587} C_VEL
LIN {X 0,Y 326.627,Z 238.795,A -85,B 0,C 180,E1 -14707.238,E2 -14707.238} C_VEL
LIN {X 0,Y 326.576,Z 238.802,A -85,B 0,C 180,E1 -14711.13,E2 -14711.13} C_VEL
LIN {X 0,Y 326.526,Z 238.806,A -85,B 0,C 180,E1 -14714.742,E2 -14714.742} C_VEL
LIN {X 0,Y 326.575,Z 238.806,A -85,B 0,C 180,E1 -14718.154,E2 -14718.154} C_VEL
LIN {X 0,Y 326.622,Z 238.797,A -85,B 0,C 180,E1 -14721.391,E2 -14721.391} C_VEL
LIN {X 0,Y 326.618,Z 238.794,A -85,B 0,C 180,E1 -14724.851,E2 -14724.851} C_VEL
LIN {X 0,Y 326.606,Z 238.798,A -85,B 0,C 180,E1 -14727.455,E2 -14727.455} C_VEL
LIN {X 0,Y 326.646,Z 238.796,A -85,B 0,C 180,E1 -14730.339,E2 -14730.339} C_VEL
LIN {X 0,Y 326.688,Z 238.787,A -85,B 0,C 180,E1 -14734.516,E2 -14734.516} C_VEL
LIN {X 0,Y 326.644,Z 238.794,A -85,B 0,C 180,E1 -14738.545,E2 -14738.545} C_VEL
LIN {X 0,Y 326.742,Z 238.781,A -85,B 0,C 180,E1 -14741.177,E2 -14741.177} C_VEL
LIN {X 0,Y 326.761,Z 238.779,A -85,B 0,C 180,E1 -14745.433,E2 -14745.433} C_VEL
LIN {X 0,Y 326.768,Z 238.774,A -85,B 0,C 180,E1 -14748.839,E2 -14748.839} C_VEL
LIN {X 0,Y 326.977,Z 238.753,A -85,B 0,C 180,E1 -14752.59,E2 -14752.59} C_VEL
LIN {X 0,Y 326.775,Z 238.777,A -85,B 0,C 180,E1 -14755.065,E2 -14755.065} C_VEL
LIN {X 0,Y 327.045,Z 238.744,A -85,B 0,C 180,E1 -14757.537,E2 -14757.537} C_VEL
LIN {X 0,Y 327.194,Z 238.728,A -85,B 0,C 180,E1 -14760,E2 -14760} C_VEL
LIN {X 0,Y 327.045,Z 238.744,A -85,B 0,C 180,E1 -14762.463,E2 -14762.463} C_VEL
LIN {X 0,Y 326.994,Z 238.755,A -85,B 0,C 180,E1 -14766.169,E2 -14766.169} C_VEL
LIN {X 0,Y 326.912,Z 238.762,A -85,B 0,C 180,E1 -14768.655,E2 -14768.655} C_VEL
LIN {X 0,Y 326.732,Z 238.783,A -85,B 0,C 180,E1 -14772.421,E2 -14772.421} C_VEL
LIN {X 0,Y 326.752,Z 238.779,A -85,B 0,C 180,E1 -14774.958,E2 -14774.958} C_VEL
LIN {X 0,Y 326.731,Z 238.784,A -85,B 0,C 180,E1 -14778.839,E2 -14778.839} C_VEL
LIN {X 0,Y 326.62,Z 238.797,A -85,B 0,C 180,E1 -14782.787,E2 -14782.787} C_VEL
LIN {X 0,Y 326.688,Z 238.788,A -85,B 0,C 180,E1 -14785.484,E2 -14785.484} C_VEL
LIN {X 0,Y 326.658,Z 238.792,A -85,B 0,C 180,E1 -14789.659,E2 -14789.659} C_VEL
LIN {X 0,Y 326.605,Z 238.8,A -85,B 0,C 180,E1 -14794.02,E2 -14794.02} C_VEL
LIN {X 0,Y 326.626,Z 238.796,A -85,B 0,C 180,E1 -14797.239,E2 -14797.239} C_VEL
LIN {X 0,Y 326.576,Z 238.802,A -85,B 0,C 180,E1 -14801.132,E2 -14801.132} C_VEL
LIN {X 0,Y 326.526,Z 238.811,A -85,B 0,C 180,E1 -14804.743,E2 -14804.743} C_VEL
LIN {X 0,Y 326.575,Z 238.806,A -85,B 0,C 180,E1 -14808.155,E2 -14808.155} C_VEL
LIN {X 0,Y 326.624,Z 238.796,A -85,B 0,C 180,E1 -14811.392,E2 -14811.392} C_VEL
LIN {X 0,Y 326.619,Z 238.801,A -85,B 0,C 180,E1 -14814.852,E2 -14814.852} C_VEL
LIN {X 0,Y 326.63,Z 238.888,A -85,B 0,C 180,E1 -14818.729,E2 -14818.729} C_VEL
LIN {X 0,Y 329.071,Z 249.932,A -85,B 0,C 180,E1 -14821.976,E2 -14821.976} C_VEL
LIN {X 0,Y 330.677,Z 258.956,A -85,B 0,C 180,E1 -14824.509,E2 -14824.509} C_VEL
LIN {X 0,Y 330.265,Z 264.789,A -85,B 0,C 180,E1 -14826.018,E2 -14826.018} C_VEL
LIN {X 0,Y 336.22,Z 302.266,A -85,B 0,C 180,E1 -14827.301,E2 -14827.301} C_VEL
LIN {X 0,Y 334.659,Z 373.389,A -85,B 0,C 180,E1 -14828.882,E2 -14828.882} C_VEL
LIN {X 0,Y 333.883,Z 387.171,A -85,B 0,C 180,E1 -14829.436,E2 -14829.436} C_VEL
LIN {X 0,Y 332.861,Z 399.591,A -85,B 0,C 180,E1 -14830.176,E2 -14830.176} C_VEL
LIN {X 0,Y 331.772,Z 411.508,A -85,B 0,C 180,E1 -14831.153,E2 -14831.153} C_VEL
LIN {X 0,Y 330.458,Z 422.957,A -85,B 0,C 180,E1 -14832.359,E2 -14832.359} C_VEL
LIN {X 0,Y 329.249,Z 433.291,A -85,B 0,C 180,E1 -14833.731,E2 -14833.731} C_VEL
LIN {X 0,Y 328.26,Z 441.738,A -85,B 0,C 180,E1 -14835.113,E2 -14835.113} C_VEL
LIN {X 0,Y 327.057,Z 450.886,A -85,B 0,C 180,E1 -14836.96,E2 -14836.96} C_VEL
LIN {X 0,Y 326.121,Z 458.252,A -85,B 0,C 180,E1 -14838.817,E2 -14838.817} C_VEL
LIN {X 0,Y 325.543,Z 464.155,A -85,B 0,C 180,E1 -14840.682,E2 -14840.682} C_VEL
LIN {X 0,Y 325.147,Z 468.794,A -85,B 0,C 180,E1 -14842.549,E2 -14842.549} C_VEL
LIN {X 0,Y 324.923,Z 472.031,A -85,B 0,C 180,E1 -14844.252,E2 -14844.252} C_VEL
LIN {X 0,Y 324.899,Z 474.811,A -85,B 0,C 180,E1 -14846.279,E2 -14846.279} C_VEL
LIN {X 0,Y 324.837,Z 475.952,A -85,B 0,C 180,E1 -14847.52,E2 -14847.52} C_VEL
LIN {X 0,Y 324.832,Z 476.659,A -85,B 0,C 180,E1 -14848.76,E2 -14848.76} C_VEL
LIN {X 0,Y 324.874,Z 476.976,A -85,B 0,C 180,E1 -14850,E2 -14850} C_VEL
LIN {X 0,Y 324.821,Z 476.901,A -85,B 0,C 180,E1 -14851.24,E2 -14851.24} C_VEL
LIN {X 0,Y 324.834,Z 476.418,A -85,B 0,C 180,E1 -14852.48,E2 -14852.48} C_VEL
LIN {X 0,Y 324.874,Z 475.504,A -85,B 0,C 180,E1 -14853.721,E2 -14853.721} C_VEL
LIN {X 0,Y 324.909,Z 473.188,A -85,B 0,C 180,E1 -14855.724,E2 -14855.724} C_VEL
LIN {X 0,Y 325.282,Z 469.041,A -85,B 0,C 180,E1 -14858.073,E2 -14858.073} C_VEL
LIN {X 0,Y 325.786,Z 464.529,A -85,B 0,C 180,E1 -14859.938,E2 -14859.938} C_VEL
LIN {X 0,Y 326.649,Z 457.713,A -85,B 0,C 180,E1 -14862.109,E2 -14862.109} C_VEL
LIN {X 0,Y 327.852,Z 450.31,A -85,B 0,C 180,E1 -14863.955,E2 -14863.955} C_VEL
LIN {X 0,Y 329.174,Z 441.138,A -85,B 0,C 180,E1 -14865.796,E2 -14865.796} C_VEL
LIN {X 0,Y 330.506,Z 431.622,A -85,B 0,C 180,E1 -14867.32,E2 -14867.32} C_VEL
LIN {X 0,Y 331.963,Z 421.091,A -85,B 0,C 180,E1 -14868.676,E2 -14868.676} C_VEL
LIN {X 0,Y 333.516,Z 409.38,A -85,B 0,C 180,E1 -14869.864,E2 -14869.864} C_VEL
LIN {X 0,Y 334.765,Z 398.013,A -85,B 0,C 180,E1 -14870.749,E2 -14870.749} C_VEL
LIN {X 0,Y 335.886,Z 384.54,A -85,B 0,C 180,E1 -14871.52,E2 -14871.52} C_VEL
LIN {X 0,Y 336.634,Z 372.088,A -85,B 0,C 180,E1 -14871.993,E2 -14871.993} C_VEL
LIN {X 0,Y 338.191,Z 302.375,A -85,B 0,C 180,E1 -14873.561,E2 -14873.561} C_VEL
LIN {X 0,Y 334.704,Z 280.626,A -85,B 0,C 180,E1 -14874.381,E2 -14874.381} C_VEL
LIN {X 0,Y 331.309,Z 263.813,A -85,B 0,C 180,E1 -14875.104,E2 -14875.104} C_VEL
LIN {X 0,Y 331.209,Z 259.987,A -85,B 0,C 180,E1 -14876.123,E2 -14876.123} C_VEL
LIN {X 0,Y 329.327,Z 250.127,A -85,B 0,C 180,E1 -14878.959,E2 -14878.959} C_VEL
LIN {X 0,Y 326.634,Z 238.803,A -85,B 0,C 180,E1 -14882.45,E2 -14882.45} C_VEL
LIN {X 0,Y 326.613,Z 238.803,A -85,B 0,C 180,E1 -14885.519,E2 -14885.519} C_VEL
LIN {X 0,Y 326.612,Z 238.802,A -85,B 0,C 180,E1 -14889.227,E2 -14889.227} C_VEL
LIN {X 0,Y 326.577,Z 238.804,A -85,B 0,C 180,E1 -14892.972,E2 -14892.972} C_VEL
LIN {X 0,Y 326.576,Z 238.808,A -85,B 0,C 180,E1 -14897.028,E2 -14897.028} C_VEL
LIN {X 0,Y 326.611,Z 238.799,A -85,B 0,C 180,E1 -14900.773,E2 -14900.773} C_VEL
LIN {X 0,Y 326.612,Z 238.796,A -85,B 0,C 180,E1 -14904.48,E2 -14904.48} C_VEL
LIN {X 0,Y 326.607,Z 238.798,A -85,B 0,C 180,E1 -14907.455,E2 -14907.455} C_VEL
LIN {X 0,Y 326.647,Z 238.794,A -85,B 0,C 180,E1 -14910.34,E2 -14910.34} C_VEL
LIN {X 0,Y 326.69,Z 238.79,A -85,B 0,C 180,E1 -14914.516,E2 -14914.516} C_VEL
LIN {X 0,Y 326.647,Z 238.794,A -85,B 0,C 180,E1 -14918.545,E2 -14918.545} C_VEL
LIN {X 0,Y 326.744,Z 238.776,A -85,B 0,C 180,E1 -14921.177,E2 -14921.177} C_VEL
LIN {X 0,Y 326.763,Z 238.771,A -85,B 0,C 180,E1 -14925.433,E2 -14925.433} C_VEL
LIN {X 0,Y 326.77,Z 238.78,A -85,B 0,C 180,E1 -14928.839,E2 -14928.839} C_VEL
LIN {X 0,Y 326.965,Z 238.756,A -85,B 0,C 180,E1 -14932.59,E2 -14932.59} C_VEL
LIN {X 0,Y 326.775,Z 238.772,A -85,B 0,C 180,E1 -14935.065,E2 -14935.065} C_VEL
LIN {X 0,Y 327.047,Z 238.746,A -85,B 0,C 180,E1 -14937.537,E2 -14937.537} C_VEL
LIN {X 0,Y 327.179,Z 238.72,A -85,B 0,C 180,E1 -14940,E2 -14940} C_VEL
LIN {X 0,Y 327.046,Z 238.748,A -85,B 0,C 180,E1 -14942.463,E2 -14942.463} C_VEL
LIN {X 0,Y 326.971,Z 238.751,A -85,B 0,C 180,E1 -14946.608,E2 -14946.608} C_VEL
LIN {X 0,Y 326.813,Z 238.774,A -85,B 0,C 180,E1 -14949.906,E2 -14949.906} C_VEL
LIN {X 0,Y 326.759,Z 238.782,A -85,B 0,C 180,E1 -14953.686,E2 -14953.686} C_VEL
LIN {X 0,Y 326.7,Z 238.788,A -85,B 0,C 180,E1 -14957.528,E2 -14957.528} C_VEL
LIN {X 0,Y 326.66,Z 238.796,A -85,B 0,C 180,E1 -14960.135,E2 -14960.135} C_VEL
LIN {X 0,Y 326.643,Z 238.795,A -85,B 0,C 180,E1 -14964.13,E2 -14964.13} C_VEL
LIN {X 0,Y 326.628,Z 238.793,A -85,B 0,C 180,E1 -14968.254,E2 -14968.254} C_VEL
LIN {X 0,Y 326.575,Z 238.805,A -85,B 0,C 180,E1 -14971.097,E2 -14971.097} C_VEL
LIN {X 0,Y 326.607,Z 238.807,A -85,B 0,C 180,E1 -14974.02,E2 -14974.02} C_VEL
LIN {X 0,Y 326.651,Z 238.903,A -85,B 0,C 180,E1 -14976.803,E2 -14976.803} C_VEL
LIN {X 0,Y 328.902,Z 248.45,A -85,B 0,C 180,E1 -14979.741,E2 -14979.741} C_VEL
LIN {X 0,Y 336.439,Z 266.619,A -85,B 0,C 180,E1 -14980.866,E2 -14980.866} C_VEL
LIN {X 0,Y 338.884,Z 279.687,A -85,B 0,C 180,E1 -14981.389,E2 -14981.389} C_VEL
LIN {X 0,Y 336.828,Z 356.039,A -85,B 0,C 180,E1 -14983.09,E2 -14983.09} C_VEL
LIN {X 0,Y 336.081,Z 369.575,A -85,B 0,C 180,E1 -14983.637,E2 -14983.637} C_VEL
LIN {X 0,Y 335.191,Z 381.617,A -85,B 0,C 180,E1 -14984.358,E2 -14984.358} C_VEL
LIN {X 0,Y 333.977,Z 394.061,A -85,B 0,C 180,E1 -14985.373,E2 -14985.373} C_VEL
LIN {X 0,Y 332.564,Z 405.814,A -85,B 0,C 180,E1 -14986.622,E2 -14986.622} C_VEL
LIN {X 0,Y 331.22,Z 415.798,A -85,B 0,C 180,E1 -14987.958,E2 -14987.958} C_VEL
LIN {X 0,Y 329.836,Z 424.899,A -85,B 0,C 180,E1 -14989.468,E2 -14989.468} C_VEL
LIN {X 0,Y 328.5,Z 433.601,A -85,B 0,C 180,E1 -14991.261,E2 -14991.261} C_VEL
LIN {X 0,Y 327.409,Z 440.61,A -85,B 0,C 180,E1 -14993.056,E2 -14993.056} C_VEL
LIN {X 0,Y 326.527,Z 446.299,A -85,B 0,C 180,E1 -14994.875,E2 -14994.875} C_VEL
LIN {X 0,Y 325.901,Z 450.661,A -85,B 0,C 180,E1 -14996.64,E2 -14996.64} C_VEL
LIN {X 0,Y 325.367,Z 454.642,A -85,B 0,C 180,E1 -14998.775,E2 -14998.775} C_VEL
LIN {X 0,Y 325.054,Z 456.514,A -85,B 0,C 180,E1 -15000.18,E2 -15000.18} C_VEL
LIN {X 0,Y 324.751,Z 458.514,A -85,B 0,C 180,E1 -15002.535,E2 -15002.535} C_VEL
LIN {X 0,Y 324.613,Z 459.041,A -85,B 0,C 180,E1 -15004.341,E2 -15004.341} C_VEL
LIN {X 0,Y 324.593,Z 458.91,A -85,B 0,C 180,E1 -15005.708,E2 -15005.708} C_VEL
LIN {X 0,Y 324.612,Z 458.261,A -85,B 0,C 180,E1 -15007.064,E2 -15007.064} C_VEL
LIN {X 0,Y 324.781,Z 457.078,A -85,B 0,C 180,E1 -15008.512,E2 -15008.512} C_VEL
LIN {X 0,Y 325.112,Z 454.62,A -85,B 0,C 180,E1 -15010.423,E2 -15010.423} C_VEL
LIN {X 0,Y 325.49,Z 450.979,A -85,B 0,C 180,E1 -15012.405,E2 -15012.405} C_VEL
LIN {X 0,Y 326.015,Z 446.132,A -85,B 0,C 180,E1 -15014.367,E2 -15014.367} C_VEL
LIN {X 0,Y 326.781,Z 439.919,A -85,B 0,C 180,E1 -15016.315,E2 -15016.315} C_VEL
LIN {X 0,Y 327.782,Z 432.147,A -85,B 0,C 180,E1 -15018.247,E2 -15018.247} C_VEL
LIN {X 0,Y 328.914,Z 423.54,A -85,B 0,C 180,E1 -15019.961,E2 -15019.961} C_VEL
LIN {X 0,Y 330.131,Z 413.329,A -85,B 0,C 180,E1 -15021.584,E2 -15021.584} C_VEL
LIN {X 0,Y 331.337,Z 403.362,A -85,B 0,C 180,E1 -15022.857,E2 -15022.857} C_VEL
LIN {X 0,Y 332.437,Z 392.92,A -85,B 0,C 180,E1 -15023.932,E2 -15023.932} C_VEL
LIN {X 0,Y 333.432,Z 381.447,A -85,B 0,C 180,E1 -15024.86,E2 -15024.86} C_VEL
LIN {X 0,Y 334.205,Z 368.607,A -85,B 0,C 180,E1 -15025.628,E2 -15025.628} C_VEL
LIN {X 0,Y 334.853,Z 355.135,A -85,B 0,C 180,E1 -15026.164,E2 -15026.164} C_VEL
LIN {X 0,Y 336.551,Z 277.506,A -85,B 0,C 180,E1 -15027.882,E2 -15027.882} C_VEL
LIN {X 0,Y 333.348,Z 261.184,A -85,B 0,C 180,E1 -15028.48,E2 -15028.48} C_VEL
LIN {X 0,Y 328.754,Z 247.932,A -85,B 0,C 180,E1 -15029.132,E2 -15029.132} C_VEL
LIN {X 0,Y 327.023,Z 238.753,A -85,B 0,C 180,E1 -15032.001,E2 -15032.001} C_VEL
LIN {X 0,Y 326.946,Z 238.76,A -85,B 0,C 180,E1 -15036.17,E2 -15036.17} C_VEL
LIN {X 0,Y 326.786,Z 238.781,A -85,B 0,C 180,E1 -15039.907,E2 -15039.907} C_VEL
LIN {X 0,Y 326.762,Z 238.784,A -85,B 0,C 180,E1 -15043.685,E2 -15043.685} C_VEL
LIN {X 0,Y 326.701,Z 238.79,A -85,B 0,C 180,E1 -15047.527,E2 -15047.527} C_VEL
LIN {X 0,Y 326.66,Z 238.795,A -85,B 0,C 180,E1 -15050.135,E2 -15050.135} C_VEL
LIN {X 0,Y 326.646,Z 238.796,A -85,B 0,C 180,E1 -15054.129,E2 -15054.129} C_VEL
LIN {X 0,Y 326.623,Z 238.797,A -85,B 0,C 180,E1 -15058.253,E2 -15058.253} C_VEL
LIN {X 0,Y 326.574,Z 238.803,A -85,B 0,C 180,E1 -15061.097,E2 -15061.097} C_VEL
LIN {X 0,Y 326.598,Z 238.798,A -85,B 0,C 180,E1 -15064.587,E2 -15064.587} C_VEL
LIN {X 0,Y 325.951,Z 238.882,A -85,B 0,C 180,E1 -15065.617,E2 -15065.617} C_VEL
LIN {X 0,Y 323.122,Z 239.235,A -85,B 0,C 180,E1 -15067.293,E2 -15067.293} C_VEL
LIN {X 0,Y 320.696,Z 239.539,A -85,B 0,C 180,E1 -15068.65,E2 -15068.65} C_VEL
LIN {X 0,Y 319.628,Z 239.671,A -85,B 0,C 180,E1 -15069.701,E2 -15069.701} C_VEL
LIN {X 0,Y 319.527,Z 239.68,A -85,B 0,C 180,E1 -15070.057,E2 -15070.057} C_VEL
LIN {X 0,Y 319.52,Z 239.68,A -85,B 0,C 180,E1 -15073.46,E2 -15073.46} C_VEL
LIN {X 0,Y 319.553,Z 239.676,A -85,B 0,C 180,E1 -15077.016,E2 -15077.016} C_VEL
LIN {X 0,Y 319.546,Z 239.679,A -85,B 0,C 180,E1 -15080.37,E2 -15080.37} C_VEL
LIN {X 0,Y 319.557,Z 239.675,A -85,B 0,C 180,E1 -15083.572,E2 -15083.572} C_VEL
LIN {X 0,Y 319.576,Z 239.673,A -85,B 0,C 180,E1 -15086.686,E2 -15086.686} C_VEL
LIN {X 0,Y 319.583,Z 239.675,A -85,B 0,C 180,E1 -15089.615,E2 -15089.615} C_VEL
LIN {X 0,Y 319.604,Z 239.671,A -85,B 0,C 180,E1 -15092.497,E2 -15092.497} C_VEL
LIN {X 0,Y 319.603,Z 239.667,A -85,B 0,C 180,E1 -15095.304,E2 -15095.304} C_VEL
LIN {X 0,Y 319.595,Z 239.673,A -85,B 0,C 180,E1 -15098.047,E2 -15098.047} C_VEL
LIN {X 0,Y 319.687,Z 239.66,A -85,B 0,C 180,E1 -15100.962,E2 -15100.962} C_VEL
LIN {X 0,Y 319.729,Z 239.654,A -85,B 0,C 180,E1 -15105.276,E2 -15105.276} C_VEL
LIN {X 0,Y 319.756,Z 239.649,A -85,B 0,C 180,E1 -15109.873,E2 -15109.873} C_VEL
LIN {X 0,Y 319.931,Z 239.632,A -85,B 0,C 180,E1 -15112.426,E2 -15112.426} C_VEL
LIN {X 0,Y 319.745,Z 239.653,A -85,B 0,C 180,E1 -15114.956,E2 -15114.956} C_VEL
LIN {X 0,Y 319.989,Z 239.623,A -85,B 0,C 180,E1 -15117.482,E2 -15117.482} C_VEL
LIN {X 0,Y 320.146,Z 239.605,A -85,B 0,C 180,E1 -15120,E2 -15120} C_VEL
LIN {X 0,Y 319.989,Z 239.622,A -85,B 0,C 180,E1 -15122.518,E2 -15122.518} C_VEL
LIN {X 0,Y 319.95,Z 239.632,A -85,B 0,C 180,E1 -15126.305,E2 -15126.305} C_VEL
LIN {X 0,Y 319.84,Z 239.642,A -85,B 0,C 180,E1 -15128.848,E2 -15128.848} C_VEL
LIN {X 0,Y 319.679,Z 239.659,A -85,B 0,C 180,E1 -15132.7,E2 -15132.7} C_VEL
LIN {X 0,Y 319.697,Z 239.657,A -85,B 0,C 180,E1 -15135.296,E2 -15135.296} C_VEL
LIN {X 0,Y 319.672,Z 239.662,A -85,B 0,C 180,E1 -15139.255,E2 -15139.255} C_VEL
LIN {X 0,Y 319.57,Z 239.674,A -85,B 0,C 180,E1 -15143.319,E2 -15143.319} C_VEL
LIN {X 0,Y 319.633,Z 239.671,A -85,B 0,C 180,E1 -15146.088,E2 -15146.088} C_VEL
LIN {X 0,Y 319.587,Z 239.673,A -85,B 0,C 180,E1 -15148.934,E2 -15148.934} C_VEL
LIN {X 0,Y 319.53,Z 239.682,A -85,B 0,C 180,E1 -15151.862,E2 -15151.862} C_VEL
LIN {X 0,Y 319.578,Z 239.674,A -85,B 0,C 180,E1 -15155.543,E2 -15155.543} C_VEL
LIN {X 0,Y 319.555,Z 239.679,A -85,B 0,C 180,E1 -15158.011,E2 -15158.011} C_VEL
LIN {X 0,Y 319.524,Z 239.68,A -85,B 0,C 180,E1 -15161.597,E2 -15161.597} C_VEL
LIN {X 0,Y 319.487,Z 239.686,A -85,B 0,C 180,E1 -15165.258,E2 -15165.258} C_VEL
LIN {X 0,Y 319.528,Z 239.684,A -85,B 0,C 180,E1 -15168.712,E2 -15168.712} C_VEL
LIN {X 0,Y 319.577,Z 239.678,A -85,B 0,C 180,E1 -15172.344,E2 -15172.344} C_VEL
LIN {X 0,Y 319.56,Z 239.68,A -85,B 0,C 180,E1 -15175.124,E2 -15175.124} C_VEL
LIN {X 0,Y 319.581,Z 239.717,A -85,B 0,C 180,E1 -15178.323,E2 -15178.323} C_VEL
LIN {X 0,Y 322.021,Z 250.792,A -85,B 0,C 180,E1 -15181.662,E2 -15181.662} C_VEL
LIN {X 0,Y 323.672,Z 259.834,A -85,B 0,C 180,E1 -15184.262,E2 -15184.262} C_VEL
LIN {X 0,Y 323.484,Z 264.594,A -85,B 0,C 180,E1 -15185.533,E2 -15185.533} C_VEL
LIN {X 0,Y 329.102,Z 300.215,A -85,B 0,C 180,E1 -15186.791,E2 -15186.791} C_VEL
LIN {X 0,Y 329.561,Z 305.391,A -85,B 0,C 180,E1 -15186.944,E2 -15186.944} C_VEL
LIN {X 0,Y 327.959,Z 373.156,A -85,B 0,C 180,E1 -15188.479,E2 -15188.479} C_VEL
LIN {X 0,Y 327.172,Z 386.8,A -85,B 0,C 180,E1 -15189.036,E2 -15189.036} C_VEL
LIN {X 0,Y 326.162,Z 398.715,A -85,B 0,C 180,E1 -15189.751,E2 -15189.751} C_VEL
LIN {X 0,Y 325.013,Z 410.821,A -85,B 0,C 180,E1 -15190.746,E2 -15190.746} C_VEL
LIN {X 0,Y 323.668,Z 422.362,A -85,B 0,C 180,E1 -15191.976,E2 -15191.976} C_VEL
LIN {X 0,Y 322.385,Z 432.772,A -85,B 0,C 180,E1 -15193.374,E2 -15193.374} C_VEL
LIN {X 0,Y 321.122,Z 442.938,A -85,B 0,C 180,E1 -15195.099,E2 -15195.099} C_VEL
LIN {X 0,Y 319.946,Z 451.856,A -85,B 0,C 180,E1 -15196.988,E2 -15196.988} C_VEL
LIN {X 0,Y 319.005,Z 458.993,A -85,B 0,C 180,E1 -15198.886,E2 -15198.886} C_VEL
LIN {X 0,Y 318.338,Z 465.498,A -85,B 0,C 180,E1 -15201.11,E2 -15201.11} C_VEL
LIN {X 0,Y 317.988,Z 469.779,A -85,B 0,C 180,E1 -15203.018,E2 -15203.018} C_VEL
LIN {X 0,Y 317.806,Z 472.976,A -85,B 0,C 180,E1 -15204.925,E2 -15204.925} C_VEL
LIN {X 0,Y 317.807,Z 474.565,A -85,B 0,C 180,E1 -15206.196,E2 -15206.196} C_VEL
LIN {X 0,Y 317.758,Z 475.728,A -85,B 0,C 180,E1 -15207.465,E2 -15207.465} C_VEL
LIN {X 0,Y 317.743,Z 476.446,A -85,B 0,C 180,E1 -15208.733,E2 -15208.733} C_VEL
LIN {X 0,Y 317.781,Z 476.774,A -85,B 0,C 180,E1 -15210,E2 -15210} C_VEL
LIN {X 0,Y 317.733,Z 476.709,A -85,B 0,C 180,E1 -15211.268,E2 -15211.268} C_VEL
LIN {X 0,Y 317.755,Z 476.246,A -85,B 0,C 180,E1 -15212.536,E2 -15212.536} C_VEL
LIN {X 0,Y 317.783,Z 475.345,A -85,B 0,C 180,E1 -15213.804,E2 -15213.804} C_VEL
LIN {X 0,Y 317.825,Z 473.288,A -85,B 0,C 180,E1 -15215.687,E2 -15215.687} C_VEL
LIN {X 0,Y 318.083,Z 470.19,A -85,B 0,C 180,E1 -15217.618,E2 -15217.618} C_VEL
LIN {X 0,Y 318.569,Z 466.073,A -85,B 0,C 180,E1 -15219.524,E2 -15219.524} C_VEL
LIN {X 0,Y 319.397,Z 459.774,A -85,B 0,C 180,E1 -15221.744,E2 -15221.744} C_VEL
LIN {X 0,Y 320.513,Z 452.934,A -85,B 0,C 180,E1 -15223.634,E2 -15223.634} C_VEL
LIN {X 0,Y 321.849,Z 444.501,A -85,B 0,C 180,E1 -15225.503,E2 -15225.503} C_VEL
LIN {X 0,Y 323.124,Z 435.711,A -85,B 0,C 180,E1 -15227.075,E2 -15227.075} C_VEL
LIN {X 0,Y 324.744,Z 424.991,A -85,B 0,C 180,E1 -15228.615,E2 -15228.615} C_VEL
LIN {X 0,Y 326.225,Z 414.356,A -85,B 0,C 180,E1 -15229.835,E2 -15229.835} C_VEL
LIN {X 0,Y 327.648,Z 402.488,A -85,B 0,C 180,E1 -15230.892,E2 -15230.892} C_VEL
LIN {X 0,Y 328.953,Z 390.192,A -85,B 0,C 180,E1 -15231.708,E2 -15231.708} C_VEL
LIN {X 0,Y 329.876,Z 377.656,A -85,B 0,C 180,E1 -15232.302,E2 -15232.302} C_VEL
LIN {X 0,Y 330.523,Z 362.586,A -85,B 0,C 180,E1 -15232.723,E2 -15232.723} C_VEL
LIN {X 0,Y 331.786,Z 303.127,A -85,B 0,C 180,E1 -15234.077,E2 -15234.077} C_VEL
LIN {X 0,Y 328.436,Z 282.161,A -85,B 0,C 180,E1 -15234.891,E2 -15234.891} C_VEL
LIN {X 0,Y 324.561,Z 263.615,A -85,B 0,C 180,E1 -15235.722,E2 -15235.722} C_VEL
LIN {X 0,Y 323.131,Z 254.947,A -85,B 0,C 180,E1 -15238.232,E2 -15238.232} C_VEL
LIN {X 0,Y 320.534,Z 243.538,A -85,B 0,C 180,E1 -15241.751,E2 -15241.751} C_VEL
LIN {X 0,Y 319.582,Z 239.68,A -85,B 0,C 180,E1 -15243.031,E2 -15243.031} C_VEL
LIN {X 0,Y 319.559,Z 239.68,A -85,B 0,C 180,E1 -15246.427,E2 -15246.427} C_VEL
LIN {X 0,Y 319.559,Z 239.677,A -85,B 0,C 180,E1 -15249.669,E2 -15249.669} C_VEL
LIN {X 0,Y 319.522,Z 239.687,A -85,B 0,C 180,E1 -15253.461,E2 -15253.461} C_VEL
LIN {X 0,Y 319.554,Z 239.683,A -85,B 0,C 180,E1 -15257.016,E2 -15257.016} C_VEL
LIN {X 0,Y 319.547,Z 239.681,A -85,B 0,C 180,E1 -15260.371,E2 -15260.371} C_VEL
LIN {X 0,Y 319.558,Z 239.678,A -85,B 0,C 180,E1 -15263.572,E2 -15263.572} C_VEL
LIN {X 0,Y 319.577,Z 239.676,A -85,B 0,C 180,E1 -15266.686,E2 -15266.686} C_VEL
LIN {X 0,Y 319.584,Z 239.673,A -85,B 0,C 180,E1 -15269.616,E2 -15269.616} C_VEL
LIN {X 0,Y 319.605,Z 239.666,A -85,B 0,C 180,E1 -15272.498,E2 -15272.498} C_VEL
LIN {X 0,Y 319.605,Z 239.672,A -85,B 0,C 180,E1 -15275.304,E2 -15275.304} C_VEL
LIN {X 0,Y 319.597,Z 239.671,A -85,B 0,C 180,E1 -15278.048,E2 -15278.048} C_VEL
LIN {X 0,Y 319.689,Z 239.656,A -85,B 0,C 180,E1 -15280.962,E2 -15280.962} C_VEL
LIN {X 0,Y 319.731,Z 239.648,A -85,B 0,C 180,E1 -15285.276,E2 -15285.276} C_VEL
LIN {X 0,Y 319.757,Z 239.647,A -85,B 0,C 180,E1 -15289.873,E2 -15289.873} C_VEL
LIN {X 0,Y 319.925,Z 239.632,A -85,B 0,C 180,E1 -15292.426,E2 -15292.426} C_VEL
LIN {X 0,Y 319.745,Z 239.648,A -85,B 0,C 180,E1 -15294.956,E2 -15294.956} C_VEL
LIN {X 0,Y 319.991,Z 239.625,A -85,B 0,C 180,E1 -15297.482,E2 -15297.482} C_VEL
LIN {X 0,Y 320.131,Z 239.598,A -85,B 0,C 180,E1 -15300,E2 -15300} C_VEL
LIN {X 0,Y 319.99,Z 239.627,A -85,B 0,C 180,E1 -15302.518,E2 -15302.518} C_VEL
LIN {X 0,Y 319.932,Z 239.63,A -85,B 0,C 180,E1 -15306.597,E2 -15306.597} C_VEL
LIN {X 0,Y 319.758,Z 239.654,A -85,B 0,C 180,E1 -15310.127,E2 -15310.127} C_VEL
LIN {X 0,Y 319.731,Z 239.655,A -85,B 0,C 180,E1 -15314.724,E2 -15314.724} C_VEL
LIN {X 0,Y 319.689,Z 239.662,A -85,B 0,C 180,E1 -15319.038,E2 -15319.038} C_VEL
LIN {X 0,Y 319.558,Z 239.677,A -85,B 0,C 180,E1 -15323.321,E2 -15323.321} C_VEL
LIN {X 0,Y 319.579,Z 239.676,A -85,B 0,C 180,E1 -15326.093,E2 -15326.093} C_VEL
LIN {X 0,Y 319.558,Z 239.67,A -85,B 0,C 180,E1 -15328.937,E2 -15328.937} C_VEL
LIN {X 0,Y 319.525,Z 239.679,A -85,B 0,C 180,E1 -15331.863,E2 -15331.863} C_VEL
LIN {X 0,Y 319.567,Z 239.68,A -85,B 0,C 180,E1 -15335.54,E2 -15335.54} C_VEL
LIN {X 0,Y 319.61,Z 239.733,A -85,B 0,C 180,E1 -15336.215,E2 -15336.215} C_VEL
LIN {X 0,Y 321.72,Z 248.639,A -85,B 0,C 180,E1 -15339.057,E2 -15339.057} C_VEL
LIN {X 0,Y 329.475,Z 266.805,A -85,B 0,C 180,E1 -15340.258,E2 -15340.258} C_VEL
LIN {X 0,Y 330.764,Z 270.823,A -85,B 0,C 180,E1 -15340.474,E2 -15340.474} C_VEL
LIN {X 0,Y 332.485,Z 280.778,A -85,B 0,C 180,E1 -15340.872,E2 -15340.872} C_VEL
LIN {X 0,Y 330.386,Z 356.034,A -85,B 0,C 180,E1 -15342.579,E2 -15342.579} C_VEL
LIN {X 0,Y 329.631,Z 369.427,A -85,B 0,C 180,E1 -15343.125,E2 -15343.125} C_VEL
LIN {X 0,Y 328.627,Z 382.29,A -85,B 0,C 180,E1 -15343.909,E2 -15343.909} C_VEL
LIN {X 0,Y 327.4,Z 394.124,A -85,B 0,C 180,E1 -15344.897,E2 -15344.897} C_VEL
LIN {X 0,Y 325.948,Z 405.795,A -85,B 0,C 180,E1 -15346.158,E2 -15346.158} C_VEL
LIN {X 0,Y 324.524,Z 415.812,A -85,B 0,C 180,E1 -15347.519,E2 -15347.519} C_VEL
LIN {X 0,Y 322.927,Z 425.882,A -85,B 0,C 180,E1 -15349.239,E2 -15349.239} C_VEL
LIN {X 0,Y 321.543,Z 434.424,A -85,B 0,C 180,E1 -15351.062,E2 -15351.062} C_VEL
LIN {X 0,Y 320.417,Z 441.341,A -85,B 0,C 180,E1 -15352.902,E2 -15352.902} C_VEL
LIN {X 0,Y 319.355,Z 447.775,A -85,B 0,C 180,E1 -15355.098,E2 -15355.098} C_VEL
LIN {X 0,Y 318.726,Z 451.906,A -85,B 0,C 180,E1 -15356.921,E2 -15356.921} C_VEL
LIN {X 0,Y 318.293,Z 455.053,A -85,B 0,C 180,E1 -15358.742,E2 -15358.742} C_VEL
LIN {X 0,Y 317.834,Z 457.597,A -85,B 0,C 180,E1 -15360.891,E2 -15360.891} C_VEL
LIN {X 0,Y 317.667,Z 458.639,A -85,B 0,C 180,E1 -15362.316,E2 -15362.316} C_VEL
LIN {X 0,Y 317.553,Z 459.176,A -85,B 0,C 180,E1 -15363.728,E2 -15363.728} C_VEL
LIN {X 0,Y 317.499,Z 459.194,A -85,B 0,C 180,E1 -15365.17,E2 -15365.17} C_VEL
LIN {X 0,Y 317.488,Z 458.78,A -85,B 0,C 180,E1 -15366.518,E2 -15366.518} C_VEL
LIN {X 0,Y 317.662,Z 457.482,A -85,B 0,C 180,E1 -15368.313,E2 -15368.313} C_VEL
LIN {X 0,Y 318.069,Z 454.599,A -85,B 0,C 180,E1 -15370.644,E2 -15370.644} C_VEL
LIN {X 0,Y 318.463,Z 450.863,A -85,B 0,C 180,E1 -15372.667,E2 -15372.667} C_VEL
LIN {X 0,Y 319.037,Z 445.911,A -85,B 0,C 180,E1 -15374.672,E2 -15374.672} C_VEL
LIN {X 0,Y 319.85,Z 439.603,A -85,B 0,C 180,E1 -15376.661,E2 -15376.661} C_VEL
LIN {X 0,Y 320.9,Z 431.727,A -85,B 0,C 180,E1 -15378.632,E2 -15378.632} C_VEL
LIN {X 0,Y 322.01,Z 423.611,A -85,B 0,C 180,E1 -15380.262,E2 -15380.262} C_VEL
LIN {X 0,Y 323.245,Z 413.665,A -85,B 0,C 180,E1 -15381.875,E2 -15381.875} C_VEL
LIN {X 0,Y 324.644,Z 402.513,A -85,B 0,C 180,E1 -15383.318,E2 -15383.318} C_VEL
LIN {X 0,Y 325.779,Z 391.37,A -85,B 0,C 180,E1 -15384.453,E2 -15384.453} C_VEL
LIN {X 0,Y 326.894,Z 378.489,A -85,B 0,C 180,E1 -15385.453,E2 -15385.453} C_VEL
LIN {X 0,Y 327.663,Z 366.049,A -85,B 0,C 180,E1 -15386.157,E2 -15386.157} C_VEL
LIN {X 0,Y 328.191,Z 353.32,A -85,B 0,C 180,E1 -15386.624,E2 -15386.624} C_VEL
LIN {X 0,Y 329.941,Z 278.574,A -85,B 0,C 180,E1 -15388.297,E2 -15388.297} C_VEL
LIN {X 0,Y 326.949,Z 263.382,A -85,B 0,C 180,E1 -15388.87,E2 -15388.87} C_VEL
LIN {X 0,Y 321.604,Z 248.13,A -85,B 0,C 180,E1 -15389.648,E2 -15389.648} C_VEL
LIN {X 0,Y 319.987,Z 239.63,A -85,B 0,C 180,E1 -15392.36,E2 -15392.36} C_VEL
LIN {X 0,Y 319.903,Z 239.637,A -85,B 0,C 180,E1 -15396.306,E2 -15396.306} C_VEL
LIN {X 0,Y 319.738,Z 239.657,A -85,B 0,C 180,E1 -15400.127,E2 -15400.127} C_VEL
LIN {X 0,Y 319.735,Z 239.66,A -85,B 0,C 180,E1 -15403.992,E2 -15403.992} C_VEL
LIN {X 0,Y 319.66,Z 239.669,A -85,B 0,C 180,E1 -15407.926,E2 -15407.926} C_VEL
LIN {X 0,Y 319.605,Z 239.671,A -85,B 0,C 180,E1 -15410.599,E2 -15410.599} C_VEL
LIN {X 0,Y 319.585,Z 239.673,A -85,B 0,C 180,E1 -15414.697,E2 -15414.697} C_VEL
LIN {X 0,Y 319.553,Z 239.675,A -85,B 0,C 180,E1 -15418.937,E2 -15418.937} C_VEL
LIN {X 0,Y 319.525,Z 239.686,A -85,B 0,C 180,E1 -15421.862,E2 -15421.862} C_VEL
LIN {X 0,Y 319.58,Z 239.674,A -85,B 0,C 180,E1 -15425.542,E2 -15425.542} C_VEL
LIN {X 0,Y 319.572,Z 239.68,A -85,B 0,C 180,E1 -15428.008,E2 -15428.008} C_VEL
LIN {X 0,Y 319.527,Z 239.68,A -85,B 0,C 180,E1 -15430.057,E2 -15430.057} C_VEL
LIN {X 0,Y 318.811,Z 239.77,A -85,B 0,C 180,E1 -15431.109,E2 -15431.109} C_VEL
LIN {X 0,Y 315.907,Z 240.129,A -85,B 0,C 180,E1 -15432.819,E2 -15432.819} C_VEL
LIN {X 0,Y 313.496,Z 240.432,A -85,B 0,C 180,E1 -15434.206,E2 -15434.206} C_VEL
LIN {X 0,Y 312.502,Z 240.553,A -85,B 0,C 180,E1 -15435.281,E2 -15435.281} C_VEL
LIN {X 0,Y 312.441,Z 240.562,A -85,B 0,C 180,E1 -15435.644,E2 -15435.644} C_VEL
LIN {X 0,Y 312.489,Z 240.557,A -85,B 0,C 180,E1 -15439.29,E2 -15439.29} C_VEL
LIN {X 0,Y 312.524,Z 240.55,A -85,B 0,C 180,E1 -15442.614,E2 -15442.614} C_VEL
LIN {X 0,Y 312.518,Z 240.554,A -85,B 0,C 180,E1 -15446.311,E2 -15446.311} C_VEL
LIN {X 0,Y 312.536,Z 240.553,A -85,B 0,C 180,E1 -15450.349,E2 -15450.349} C_VEL
LIN {X 0,Y 312.601,Z 240.544,A -85,B 0,C 180,E1 -15454.064,E2 -15454.064} C_VEL
LIN {X 0,Y 312.585,Z 240.541,A -85,B 0,C 180,E1 -15457.529,E2 -15457.529} C_VEL
LIN {X 0,Y 312.636,Z 240.54,A -85,B 0,C 180,E1 -15461.656,E2 -15461.656} C_VEL
LIN {X 0,Y 312.692,Z 240.532,A -85,B 0,C 180,E1 -15465.686,E2 -15465.686} C_VEL
LIN {X 0,Y 312.7,Z 240.524,A -85,B 0,C 180,E1 -15469.642,E2 -15469.642} C_VEL
LIN {X 0,Y 312.87,Z 240.513,A -85,B 0,C 180,E1 -15472.254,E2 -15472.254} C_VEL
LIN {X 0,Y 312.716,Z 240.529,A -85,B 0,C 180,E1 -15474.842,E2 -15474.842} C_VEL
LIN {X 0,Y 312.988,Z 240.494,A -85,B 0,C 180,E1 -15478.713,E2 -15478.713} C_VEL
LIN {X 0,Y 312.986,Z 240.489,A -85,B 0,C 180,E1 -15481.287,E2 -15481.287} C_VEL
LIN {X 0,Y 312.716,Z 240.527,A -85,B 0,C 180,E1 -15485.158,E2 -15485.158} C_VEL
LIN {X 0,Y 312.87,Z 240.511,A -85,B 0,C 180,E1 -15487.746,E2 -15487.746} C_VEL
LIN {X 0,Y 312.667,Z 240.534,A -85,B 0,C 180,E1 -15491.671,E2 -15491.671} C_VEL
LIN {X 0,Y 312.697,Z 240.529,A -85,B 0,C 180,E1 -15494.888,E2 -15494.888} C_VEL
LIN {X 0,Y 312.628,Z 240.54,A -85,B 0,C 180,E1 -15499.237,E2 -15499.237} C_VEL
LIN {X 0,Y 312.544,Z 240.55,A -85,B 0,C 180,E1 -15502.79,E2 -15502.79} C_VEL
LIN {X 0,Y 312.601,Z 240.545,A -85,B 0,C 180,E1 -15505.936,E2 -15505.936} C_VEL
LIN {X 0,Y 312.543,Z 240.55,A -85,B 0,C 180,E1 -15509.65,E2 -15509.65} C_VEL
LIN {X 0,Y 312.517,Z 240.553,A -85,B 0,C 180,E1 -15513.689,E2 -15513.689} C_VEL
LIN {X 0,Y 312.524,Z 240.552,A -85,B 0,C 180,E1 -15517.385,E2 -15517.385} C_VEL
LIN {X 0,Y 312.488,Z 240.559,A -85,B 0,C 180,E1 -15520.71,E2 -15520.71} C_VEL
LIN {X 0,Y 312.45,Z 240.564,A -85,B 0,C 180,E1 -15524.21,E2 -15524.21} C_VEL
LIN {X 0,Y 312.512,Z 240.556,A -85,B 0,C 180,E1 -15527.913,E2 -15527.913} C_VEL
LIN {X 0,Y 312.535,Z 240.552,A -85,B 0,C 180,E1 -15531.911,E2 -15531.911} C_VEL
LIN {X 0,Y 312.506,Z 240.559,A -85,B 0,C 180,E1 -15535.79,E2 -15535.79} C_VEL
LIN {X 0,Y 312.557,Z 240.703,A -85,B 0,C 180,E1 -15537.952,E2 -15537.952} C_VEL
LIN {X 0,Y 314.979,Z 251.642,A -85,B 0,C 180,E1 -15541.333,E2 -15541.333} C_VEL
LIN {X 0,Y 316.816,Z 261.978,A -85,B 0,C 180,E1 -15544.369,E2 -15544.369} C_VEL
LIN {X 0,Y 316.691,Z 264.362,A -85,B 0,C 180,E1 -15545.018,E2 -15545.018} C_VEL
LIN {X 0,Y 322.32,Z 299.742,A -85,B 0,C 180,E1 -15546.318,E2 -15546.318} C_VEL
LIN {X 0,Y 322.934,Z 305.514,A -85,B 0,C 180,E1 -15546.501,E2 -15546.501} C_VEL
LIN {X 0,Y 321.299,Z 372.839,A -85,B 0,C 180,E1 -15548.057,E2 -15548.057} C_VEL
LIN {X 0,Y 320.552,Z 385.674,A -85,B 0,C 180,E1 -15548.582,E2 -15548.582} C_VEL
LIN {X 0,Y 319.372,Z 398.946,A -85,B 0,C 180,E1 -15549.385,E2 -15549.385} C_VEL
LIN {X 0,Y 318.258,Z 410.133,A -85,B 0,C 180,E1 -15550.321,E2 -15550.321} C_VEL
LIN {X 0,Y 316.871,Z 421.765,A -85,B 0,C 180,E1 -15551.576,E2 -15551.576} C_VEL
LIN {X 0,Y 315.55,Z 432.246,A -85,B 0,C 180,E1 -15553.003,E2 -15553.003} C_VEL
LIN {X 0,Y 314.511,Z 440.819,A -85,B 0,C 180,E1 -15554.446,E2 -15554.446} C_VEL
LIN {X 0,Y 313.409,Z 448.71,A -85,B 0,C 180,E1 -15556.051,E2 -15556.051} C_VEL
LIN {X 0,Y 312.278,Z 456.399,A -85,B 0,C 180,E1 -15557.985,E2 -15557.985} C_VEL
LIN {X 0,Y 311.441,Z 463.495,A -85,B 0,C 180,E1 -15560.256,E2 -15560.256} C_VEL
LIN {X 0,Y 311.01,Z 468.196,A -85,B 0,C 180,E1 -15562.208,E2 -15562.208} C_VEL
LIN {X 0,Y 310.729,Z 472.109,A -85,B 0,C 180,E1 -15564.375,E2 -15564.375} C_VEL
LIN {X 0,Y 310.717,Z 474.315,A -85,B 0,C 180,E1 -15566.109,E2 -15566.109} C_VEL
LIN {X 0,Y 310.682,Z 475.499,A -85,B 0,C 180,E1 -15567.407,E2 -15567.407} C_VEL
LIN {X 0,Y 310.658,Z 476.232,A -85,B 0,C 180,E1 -15568.704,E2 -15568.704} C_VEL
LIN {X 0,Y 310.691,Z 476.571,A -85,B 0,C 180,E1 -15570,E2 -15570} C_VEL
LIN {X 0,Y 310.648,Z 476.518,A -85,B 0,C 180,E1 -15571.297,E2 -15571.297} C_VEL
LIN {X 0,Y 310.677,Z 476.072,A -85,B 0,C 180,E1 -15572.593,E2 -15572.593} C_VEL
LIN {X 0,Y 310.696,Z 475.187,A -85,B 0,C 180,E1 -15573.891,E2 -15573.891} C_VEL
LIN {X 0,Y 310.821,Z 472.205,A -85,B 0,C 180,E1 -15576.492,E2 -15576.492} C_VEL
LIN {X 0,Y 311.186,Z 468.814,A -85,B 0,C 180,E1 -15578.442,E2 -15578.442} C_VEL
LIN {X 0,Y 311.742,Z 464.35,A -85,B 0,C 180,E1 -15580.391,E2 -15580.391} C_VEL
LIN {X 0,Y 312.72,Z 457.618,A -85,B 0,C 180,E1 -15582.657,E2 -15582.657} C_VEL
LIN {X 0,Y 314.074,Z 450.288,A -85,B 0,C 180,E1 -15584.581,E2 -15584.581} C_VEL
LIN {X 0,Y 315.554,Z 440.98,A -85,B 0,C 180,E1 -15586.545,E2 -15586.545} C_VEL
LIN {X 0,Y 317.121,Z 430.777,A -85,B 0,C 180,E1 -15588.242,E2 -15588.242} C_VEL
LIN {X 0,Y 318.792,Z 420.168,A -85,B 0,C 180,E1 -15589.645,E2 -15589.645} C_VEL
LIN {X 0,Y 320.241,Z 409.951,A -85,B 0,C 180,E1 -15590.725,E2 -15590.725} C_VEL
LIN {X 0,Y 321.582,Z 398.958,A -85,B 0,C 180,E1 -15591.641,E2 -15591.641} C_VEL
LIN {X 0,Y 322.791,Z 386.027,A -85,B 0,C 180,E1 -15592.439,E2 -15592.439} C_VEL
LIN {X 0,Y 323.718,Z 372.315,A -85,B 0,C 180,E1 -15593.003,E2 -15593.003} C_VEL
LIN {X 0,Y 325.47,Z 304.42,A -85,B 0,C 180,E1 -15594.594,E2 -15594.594} C_VEL
LIN {X 0,Y 322.184,Z 283.625,A -85,B 0,C 180,E1 -15595.427,E2 -15595.427} C_VEL
LIN {X 0,Y 318.558,Z 266.313,A -85,B 0,C 180,E1 -15596.232,E2 -15596.232} C_VEL
LIN {X 0,Y 317.512,Z 263.336,A -85,B 0,C 180,E1 -15596.429,E2 -15596.429} C_VEL
LIN {X 0,Y 315.672,Z 253.734,A -85,B 0,C 180,E1 -15599.327,E2 -15599.327} C_VEL
LIN {X 0,Y 312.993,Z 242.498,A -85,B 0,C 180,E1 -15602.952,E2 -15602.952} C_VEL
LIN {X 0,Y 312.513,Z 240.563,A -85,B 0,C 180,E1 -15603.619,E2 -15603.619} C_VEL
LIN {X 0,Y 312.526,Z 240.556,A -85,B 0,C 180,E1 -15607.385,E2 -15607.385} C_VEL
LIN {X 0,Y 312.491,Z 240.559,A -85,B 0,C 180,E1 -15610.709,E2 -15610.709} C_VEL
LIN {X 0,Y 312.452,Z 240.566,A -85,B 0,C 180,E1 -15614.209,E2 -15614.209} C_VEL
LIN {X 0,Y 312.484,Z 240.555,A -85,B 0,C 180,E1 -15617.919,E2 -15617.919} C_VEL
LIN {X 0,Y 312.505,Z 240.555,A -85,B 0,C 180,E1 -15621.917,E2 -15621.917} C_VEL
LIN {X 0,Y 312.532,Z 240.551,A -85,B 0,C 180,E1 -15624.22,E2 -15624.22} C_VEL
LIN {X 0,Y 312.503,Z 240.555,A -85,B 0,C 180,E1 -15627.334,E2 -15627.334} C_VEL
LIN {X 0,Y 312.544,Z 240.55,A -85,B 0,C 180,E1 -15631.279,E2 -15631.279} C_VEL
LIN {X 0,Y 312.585,Z 240.548,A -85,B 0,C 180,E1 -15634.711,E2 -15634.711} C_VEL
LIN {X 0,Y 312.587,Z 240.542,A -85,B 0,C 180,E1 -15637.529,E2 -15637.529} C_VEL
LIN {X 0,Y 312.638,Z 240.532,A -85,B 0,C 180,E1 -15641.656,E2 -15641.656} C_VEL
LIN {X 0,Y 312.693,Z 240.522,A -85,B 0,C 180,E1 -15645.686,E2 -15645.686} C_VEL
LIN {X 0,Y 312.701,Z 240.526,A -85,B 0,C 180,E1 -15649.642,E2 -15649.642} C_VEL
LIN {X 0,Y 312.865,Z 240.51,A -85,B 0,C 180,E1 -15652.254,E2 -15652.254} C_VEL
LIN {X 0,Y 312.715,Z 240.523,A -85,B 0,C 180,E1 -15654.842,E2 -15654.842} C_VEL
LIN {X 0,Y 312.988,Z 240.493,A -85,B 0,C 180,E1 -15658.713,E2 -15658.713} C_VEL
LIN {X 0,Y 312.99,Z 240.498,A -85,B 0,C 180,E1 -15661.287,E2 -15661.287} C_VEL
LIN {X 0,Y 312.715,Z 240.53,A -85,B 0,C 180,E1 -15665.158,E2 -15665.158} C_VEL
LIN {X 0,Y 312.871,Z 240.505,A -85,B 0,C 180,E1 -15667.746,E2 -15667.746} C_VEL
LIN {X 0,Y 312.669,Z 240.53,A -85,B 0,C 180,E1 -15671.671,E2 -15671.671} C_VEL
LIN {X 0,Y 312.7,Z 240.529,A -85,B 0,C 180,E1 -15674.888,E2 -15674.888} C_VEL
LIN {X 0,Y 312.629,Z 240.543,A -85,B 0,C 180,E1 -15679.236,E2 -15679.236} C_VEL
LIN {X 0,Y 312.525,Z 240.557,A -85,B 0,C 180,E1 -15682.78,E2 -15682.78} C_VEL
LIN {X 0,Y 312.538,Z 240.553,A -85,B 0,C 180,E1 -15685.911,E2 -15685.911} C_VEL
LIN {X 0,Y 312.504,Z 240.55,A -85,B 0,C 180,E1 -15689.655,E2 -15689.655} C_VEL
LIN {X 0,Y 312.52,Z 240.561,A -85,B 0,C 180,E1 -15693.689,E2 -15693.689} C_VEL
LIN {X 0,Y 312.545,Z 240.672,A -85,B 0,C 180,E1 -15695.629,E2 -15695.629} C_VEL
LIN {X 0,Y 314.526,Z 248.792,A -85,B 0,C 180,E1 -15698.333,E2 -15698.333} C_VEL
LIN {X 0,Y 322.769,Z 267.549,A -85,B 0,C 180,E1 -15699.653,E2 -15699.653} C_VEL
LIN {X 0,Y 324.678,Z 273.213,A -85,B 0,C 180,E1 -15699.98,E2 -15699.98} C_VEL
LIN {X 0,Y 326.154,Z 280.991,A -85,B 0,C 180,E1 -15700.315,E2 -15700.315} C_VEL
LIN {X 0,Y 323.934,Z 356.708,A -85,B 0,C 180,E1 -15702.07,E2 -15702.07} C_VEL
LIN {X 0,Y 323.142,Z 370.044,A -85,B 0,C 180,E1 -15702.632,E2 -15702.632} C_VEL
LIN {X 0,Y 322.149,Z 382.179,A -85,B 0,C 180,E1 -15703.386,E2 -15703.386} C_VEL
LIN {X 0,Y 320.935,Z 393.727,A -85,B 0,C 180,E1 -15704.356,E2 -15704.356} C_VEL
LIN {X 0,Y 319.35,Z 405.81,A -85,B 0,C 180,E1 -15705.675,E2 -15705.675} C_VEL
LIN {X 0,Y 317.758,Z 416.53,A -85,B 0,C 180,E1 -15707.165,E2 -15707.165} C_VEL
LIN {X 0,Y 316.238,Z 425.712,A -85,B 0,C 180,E1 -15708.766,E2 -15708.766} C_VEL
LIN {X 0,Y 314.861,Z 433.758,A -85,B 0,C 180,E1 -15710.495,E2 -15710.495} C_VEL
LIN {X 0,Y 313.592,Z 441.058,A -85,B 0,C 180,E1 -15712.44,E2 -15712.44} C_VEL
LIN {X 0,Y 312.62,Z 446.445,A -85,B 0,C 180,E1 -15714.232,E2 -15714.232} C_VEL
LIN {X 0,Y 311.752,Z 451.789,A -85,B 0,C 180,E1 -15716.524,E2 -15716.524} C_VEL
LIN {X 0,Y 311.204,Z 455.462,A -85,B 0,C 180,E1 -15718.707,E2 -15718.707} C_VEL
LIN {X 0,Y 310.857,Z 457.251,A -85,B 0,C 180,E1 -15720.173,E2 -15720.173} C_VEL
LIN {X 0,Y 310.62,Z 458.673,A -85,B 0,C 180,E1 -15721.934,E2 -15721.934} C_VEL
LIN {X 0,Y 310.41,Z 459.466,A -85,B 0,C 180,E1 -15724.521,E2 -15724.521} C_VEL
LIN {X 0,Y 310.401,Z 459.19,A -85,B 0,C 180,E1 -15725.949,E2 -15725.949} C_VEL
LIN {X 0,Y 310.529,Z 457.878,A -85,B 0,C 180,E1 -15728.115,E2 -15728.115} C_VEL
LIN {X 0,Y 311.009,Z 454.554,A -85,B 0,C 180,E1 -15730.874,E2 -15730.874} C_VEL
LIN {X 0,Y 311.435,Z 450.732,A -85,B 0,C 180,E1 -15732.94,E2 -15732.94} C_VEL
LIN {X 0,Y 312.052,Z 445.777,A -85,B 0,C 180,E1 -15734.959,E2 -15734.959} C_VEL
LIN {X 0,Y 312.919,Z 439.29,A -85,B 0,C 180,E1 -15737.021,E2 -15737.021} C_VEL
LIN {X 0,Y 313.844,Z 432.584,A -85,B 0,C 180,E1 -15738.733,E2 -15738.733} C_VEL
LIN {X 0,Y 314.985,Z 424.78,A -85,B 0,C 180,E1 -15740.367,E2 -15740.367} C_VEL
LIN {X 0,Y 316.26,Z 415.095,A -85,B 0,C 180,E1 -15742.016,E2 -15742.016} C_VEL
LIN {X 0,Y 317.66,Z 404.21,A -85,B 0,C 180,E1 -15743.489,E2 -15743.489} C_VEL
LIN {X 0,Y 318.886,Z 393.225,A -85,B 0,C 180,E1 -15744.673,E2 -15744.673} C_VEL
LIN {X 0,Y 319.977,Z 381.274,A -85,B 0,C 180,E1 -15745.67,E2 -15745.67} C_VEL
LIN {X 0,Y 320.84,Z 368.21,A -85,B 0,C 180,E1 -15746.468,E2 -15746.468} C_VEL
LIN {X 0,Y 321.47,Z 355.556,A -85,B 0,C 180,E1 -15746.984,E2 -15746.984} C_VEL
LIN {X 0,Y 323.37,Z 279.675,A -85,B 0,C 180,E1 -15748.727,E2 -15748.727} C_VEL
LIN {X 0,Y 320.483,Z 265.245,A -85,B 0,C 180,E1 -15749.289,E2 -15749.289} C_VEL
LIN {X 0,Y 314.442,Z 248.274,A -85,B 0,C 180,E1 -15750.2,E2 -15750.2} C_VEL
LIN {X 0,Y 312.849,Z 240.518,A -85,B 0,C 180,E1 -15752.776,E2 -15752.776} C_VEL
LIN {X 0,Y 312.844,Z 240.516,A -85,B 0,C 180,E1 -15756.449,E2 -15756.449} C_VEL
LIN {X 0,Y 312.753,Z 240.526,A -85,B 0,C 180,E1 -15759.05,E2 -15759.05} C_VEL
LIN {X 0,Y 312.637,Z 240.54,A -85,B 0,C 180,E1 -15762.991,E2 -15762.991} C_VEL
LIN {X 0,Y 312.64,Z 240.544,A -85,B 0,C 180,E1 -15765.649,E2 -15765.649} C_VEL
LIN {X 0,Y 312.631,Z 240.541,A -85,B 0,C 180,E1 -15769.235,E2 -15769.235} C_VEL
LIN {X 0,Y 312.528,Z 240.55,A -85,B 0,C 180,E1 -15772.78,E2 -15772.78} C_VEL
LIN {X 0,Y 312.537,Z 240.556,A -85,B 0,C 180,E1 -15775.91,E2 -15775.91} C_VEL
LIN {X 0,Y 312.501,Z 240.557,A -85,B 0,C 180,E1 -15779.654,E2 -15779.654} C_VEL
LIN {X 0,Y 312.52,Z 240.557,A -85,B 0,C 180,E1 -15783.688,E2 -15783.688} C_VEL
LIN {X 0,Y 312.525,Z 240.552,A -85,B 0,C 180,E1 -15787.385,E2 -15787.385} C_VEL
LIN {X 0,Y 312.489,Z 240.557,A -85,B 0,C 180,E1 -15790.709,E2 -15790.709} C_VEL
LIN {X 0,Y 312.451,Z 240.562,A -85,B 0,C 180,E1 -15794.209,E2 -15794.209} C_VEL
LIN {X 0,Y 312.441,Z 240.562,A -85,B 0,C 180,E1 -15795.644,E2 -15795.644} C_VEL
LIN {X 0,Y 311.816,Z 240.645,A -85,B 0,C 180,E1 -15796.721,E2 -15796.721} C_VEL
LIN {X 0,Y 308.952,Z 241,A -85,B 0,C 180,E1 -15798.474,E2 -15798.474} C_VEL
LIN {X 0,Y 306.522,Z 241.305,A -85,B 0,C 180,E1 -15799.896,E2 -15799.896} C_VEL
LIN {X 0,Y 305.518,Z 241.425,A -85,B 0,C 180,E1 -15800.997,E2 -15800.997} C_VEL
LIN {X 0,Y 305.458,Z 241.432,A -85,B 0,C 180,E1 -15801.37,E2 -15801.37} C_VEL
LIN {X 0,Y 305.461,Z 241.426,A -85,B 0,C 180,E1 -15804.886,E2 -15804.886} C_VEL
LIN {X 0,Y 305.448,Z 241.436,A -85,B 0,C 180,E1 -15808.355,E2 -15808.355} C_VEL
LIN {X 0,Y 305.511,Z 241.426,A -85,B 0,C 180,E1 -15811.113,E2 -15811.113} C_VEL
LIN {X 0,Y 305.569,Z 241.418,A -85,B 0,C 180,E1 -15814.087,E2 -15814.087} C_VEL
LIN {X 0,Y 305.498,Z 241.428,A -85,B 0,C 180,E1 -15818.402,E2 -15818.402} C_VEL
LIN {X 0,Y 305.588,Z 241.416,A -85,B 0,C 180,E1 -15821.217,E2 -15821.217} C_VEL
LIN {X 0,Y 305.647,Z 241.408,A -85,B 0,C 180,E1 -15825.349,E2 -15825.349} C_VEL
LIN {X 0,Y 305.636,Z 241.402,A -85,B 0,C 180,E1 -15829.399,E2 -15829.399} C_VEL
LIN {X 0,Y 305.811,Z 241.39,A -85,B 0,C 180,E1 -15832.074,E2 -15832.074} C_VEL
